REGION Network 61: UNIT 2 STATION 3 MEASURING RESET METHOD WORKING OR BLOCKED ALARM
   RUNG wire#powerrail
      Contact( "DB16337_U2_STA3_MEAS_RESET_TRIG".Done )
      I_Contact( "DB16004_U2_STA3_MEAS_CLIENT_INTERFACE".U02_STA3_MEAS_Method."Trigger reset".Outputs.Result )
      wire#w1
      Contact( "DB7256_UNIT_2_STA_3_MEAS_ENABLE_DISABLE".ENABLED )
      wire#w2
      Coil( "DB16000_OPC_UA_TRIGGER_ALARM".CLIENT.U2_STA3_MEAS.ALARMS.RESET_METHOD_WORKING_BLOCKED_A )
   END_RUNG
   RUNG wire#powerrail
      Contact( "DB16000_OPC_UA_TRIGGER_ALARM".CLIENT.U2_STA3_MEAS.ALARMS.RESET_METHOD_WORKING_BLOCKED_A )
      I_Contact( "DB2120_MPP_ITC_IPC".RESET_FAULTS )
   END_RUNG wire#w1
   RUNG wire#w2
      Coil( "DB426_ALARMS_WARNINGS".ALARMS.UNIT_02.STATION_3_MEASURING."720731" )
   END_RUNG
   // the same network as SCL:
   "DB16000_OPC_UA_TRIGGER_ALARM".CLIENT.U2_STA3_MEAS.ALARMS.RESET_METHOD_WORKING_BLOCKED_A := (("DB16337_U2_STA3_MEAS_RESET_TRIG".Done AND NOT "DB16004_U2_STA3_MEAS_CLIENT_INTERFACE".U02_STA3_MEAS_Method."Trigger reset".Outputs.Result) OR ("DB16000_OPC_UA_TRIGGER_ALARM".CLIENT.U2_STA3_MEAS.ALARMS.RESET_METHOD_WORKING_BLOCKED_A AND NOT "DB2120_MPP_ITC_IPC".RESET_FAULTS)) AND "DB7256_UNIT_2_STA_3_MEAS_ENABLE_DISABLE".ENABLED;
   "DB426_ALARMS_WARNINGS".ALARMS.UNIT_02.STATION_3_MEASURING."720731" := "DB16000_OPC_UA_TRIGGER_ALARM".CLIENT.U2_STA3_MEAS.ALARMS.RESET_METHOD_WORKING_BLOCKED_A;
END_REGION

REGION Network 62: UNIT 2 STATION 3 MEASURING READ VARIABLES CONNECTION ALARM
   RUNG wire#powerrail
      Contact( "DB16330_READLIST_U2_STA3_MEAS".Error )
      wire#w1
      Contact( "DB7256_UNIT_2_STA_3_MEAS_ENABLE_DISABLE".ENABLED )
      wire#w2
      Coil( "DB16000_OPC_UA_TRIGGER_ALARM".CLIENT.U2_STA3_MEAS.ALARMS.READ_VAR_CONNECTION_A )
   END_RUNG
   RUNG wire#powerrail
      Contact( "DB16000_OPC_UA_TRIGGER_ALARM".CLIENT.U2_STA3_MEAS.ALARMS.READ_VAR_CONNECTION_A )
      I_Contact( "DB2120_MPP_ITC_IPC".RESET_FAULTS )
   END_RUNG wire#w1
   RUNG wire#w2
      Coil( "DB426_ALARMS_WARNINGS".ALARMS.UNIT_02.STATION_3_MEASURING."720738" )
   END_RUNG
   // the same network as SCL:
   "DB16000_OPC_UA_TRIGGER_ALARM".CLIENT.U2_STA3_MEAS.ALARMS.READ_VAR_CONNECTION_A := ("DB16330_READLIST_U2_STA3_MEAS".Error OR ("DB16000_OPC_UA_TRIGGER_ALARM".CLIENT.U2_STA3_MEAS.ALARMS.READ_VAR_CONNECTION_A AND NOT "DB2120_MPP_ITC_IPC".RESET_FAULTS)) AND "DB7256_UNIT_2_STA_3_MEAS_ENABLE_DISABLE".ENABLED;
   "DB426_ALARMS_WARNINGS".ALARMS.UNIT_02.STATION_3_MEASURING."720738" := "DB16000_OPC_UA_TRIGGER_ALARM".CLIENT.U2_STA3_MEAS.ALARMS.READ_VAR_CONNECTION_A;
END_REGION

REGION Network 63: UNIT 2 STATION 3 MEASURING READ VARIABLES WORKING OR BLOCKED ALARM
   RUNG wire#powerrail
      Contact( "DB16330_READLIST_U2_STA3_MEAS".Done )
      Contact( "M_DUMMY_OFF" )
      wire#w1
      Contact( "DB7256_UNIT_2_STA_3_MEAS_ENABLE_DISABLE".ENABLED )
      wire#w2
      Coil( "DB16000_OPC_UA_TRIGGER_ALARM".CLIENT.U2_STA3_MEAS.ALARMS.READ_VAR_METHOD_WORKING_BLOCKED_A )
   END_RUNG
   RUNG wire#powerrail
      Contact( "DB16000_OPC_UA_TRIGGER_ALARM".CLIENT.U2_STA3_MEAS.ALARMS.READ_VAR_METHOD_WORKING_BLOCKED_A )
      I_Contact( "DB2120_MPP_ITC_IPC".RESET_FAULTS )
   END_RUNG wire#w1
   RUNG wire#w2
      Coil( "DB426_ALARMS_WARNINGS".ALARMS.UNIT_02.STATION_3_MEASURING."720739" )
   END_RUNG
   // the same network as SCL:
   "DB16000_OPC_UA_TRIGGER_ALARM".CLIENT.U2_STA3_MEAS.ALARMS.READ_VAR_METHOD_WORKING_BLOCKED_A := (("DB16330_READLIST_U2_STA3_MEAS".Done AND "M_DUMMY_OFF") OR ("DB16000_OPC_UA_TRIGGER_ALARM".CLIENT.U2_STA3_MEAS.ALARMS.READ_VAR_METHOD_WORKING_BLOCKED_A AND NOT "DB2120_MPP_ITC_IPC".RESET_FAULTS)) AND "DB7256_UNIT_2_STA_3_MEAS_ENABLE_DISABLE".ENABLED;
   "DB426_ALARMS_WARNINGS".ALARMS.UNIT_02.STATION_3_MEASURING."720739" := "DB16000_OPC_UA_TRIGGER_ALARM".CLIENT.U2_STA3_MEAS.ALARMS.READ_VAR_METHOD_WORKING_BLOCKED_A;
END_REGION

REGION Network 64: UNIT 2 STATION 3 MEASURING PROFILER CONFIGURATION ALARM
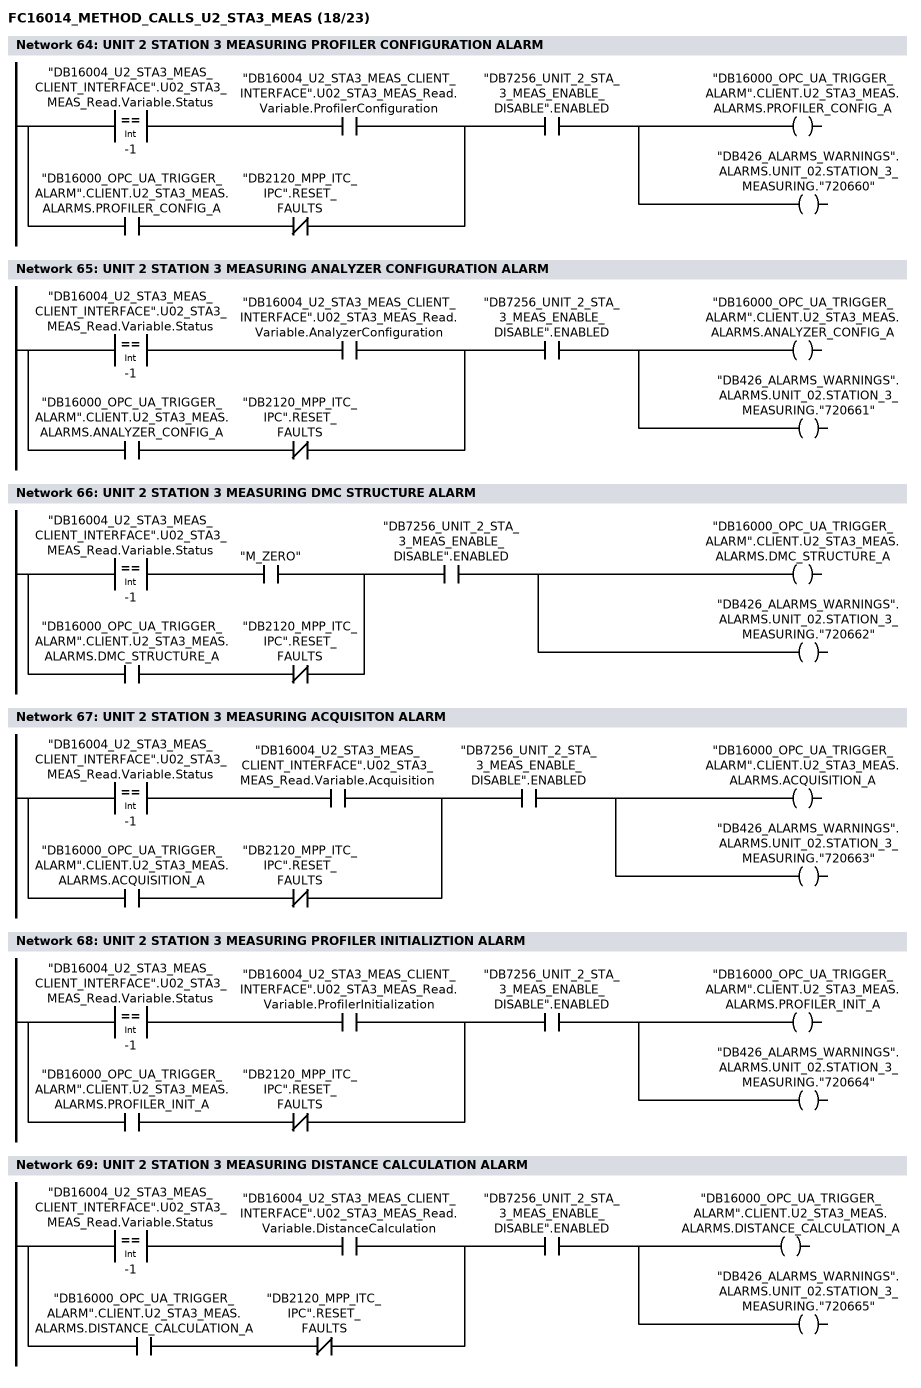
   RUNG wire#powerrail
      { S7_Templates := "SrcType := Int" } EQ_Contact(in1 := "DB16004_U2_STA3_MEAS_CLIENT_INTERFACE".U02_STA3_MEAS_Read.Variable.Status, in2 := -1)
      Contact( "DB16004_U2_STA3_MEAS_CLIENT_INTERFACE".U02_STA3_MEAS_Read.Variable.ProfilerConfiguration )
      wire#w1
      Contact( "DB7256_UNIT_2_STA_3_MEAS_ENABLE_DISABLE".ENABLED )
      wire#w2
      Coil( "DB16000_OPC_UA_TRIGGER_ALARM".CLIENT.U2_STA3_MEAS.ALARMS.PROFILER_CONFIG_A )
   END_RUNG
   RUNG wire#powerrail
      Contact( "DB16000_OPC_UA_TRIGGER_ALARM".CLIENT.U2_STA3_MEAS.ALARMS.PROFILER_CONFIG_A )
      I_Contact( "DB2120_MPP_ITC_IPC".RESET_FAULTS )
   END_RUNG wire#w1
   RUNG wire#w2
      Coil( "DB426_ALARMS_WARNINGS".ALARMS.UNIT_02.STATION_3_MEASURING."720660" )
   END_RUNG
   // the same network as SCL:
   "DB16000_OPC_UA_TRIGGER_ALARM".CLIENT.U2_STA3_MEAS.ALARMS.PROFILER_CONFIG_A := ((("DB16004_U2_STA3_MEAS_CLIENT_INTERFACE".U02_STA3_MEAS_Read.Variable.Status = (-1)) AND "DB16004_U2_STA3_MEAS_CLIENT_INTERFACE".U02_STA3_MEAS_Read.Variable.ProfilerConfiguration) OR ("DB16000_OPC_UA_TRIGGER_ALARM".CLIENT.U2_STA3_MEAS.ALARMS.PROFILER_CONFIG_A AND NOT "DB2120_MPP_ITC_IPC".RESET_FAULTS)) AND "DB7256_UNIT_2_STA_3_MEAS_ENABLE_DISABLE".ENABLED;
   "DB426_ALARMS_WARNINGS".ALARMS.UNIT_02.STATION_3_MEASURING."720660" := "DB16000_OPC_UA_TRIGGER_ALARM".CLIENT.U2_STA3_MEAS.ALARMS.PROFILER_CONFIG_A;
END_REGION

REGION Network 65: UNIT 2 STATION 3 MEASURING ANALYZER CONFIGURATION ALARM
   RUNG wire#powerrail
      { S7_Templates := "SrcType := Int" } EQ_Contact(in1 := "DB16004_U2_STA3_MEAS_CLIENT_INTERFACE".U02_STA3_MEAS_Read.Variable.Status, in2 := -1)
      Contact( "DB16004_U2_STA3_MEAS_CLIENT_INTERFACE".U02_STA3_MEAS_Read.Variable.AnalyzerConfiguration )
      wire#w1
      Contact( "DB7256_UNIT_2_STA_3_MEAS_ENABLE_DISABLE".ENABLED )
      wire#w2
      Coil( "DB16000_OPC_UA_TRIGGER_ALARM".CLIENT.U2_STA3_MEAS.ALARMS.ANALYZER_CONFIG_A )
   END_RUNG
   RUNG wire#powerrail
      Contact( "DB16000_OPC_UA_TRIGGER_ALARM".CLIENT.U2_STA3_MEAS.ALARMS.ANALYZER_CONFIG_A )
      I_Contact( "DB2120_MPP_ITC_IPC".RESET_FAULTS )
   END_RUNG wire#w1
   RUNG wire#w2
      Coil( "DB426_ALARMS_WARNINGS".ALARMS.UNIT_02.STATION_3_MEASURING."720661" )
   END_RUNG
   // the same network as SCL:
   "DB16000_OPC_UA_TRIGGER_ALARM".CLIENT.U2_STA3_MEAS.ALARMS.ANALYZER_CONFIG_A := ((("DB16004_U2_STA3_MEAS_CLIENT_INTERFACE".U02_STA3_MEAS_Read.Variable.Status = (-1)) AND "DB16004_U2_STA3_MEAS_CLIENT_INTERFACE".U02_STA3_MEAS_Read.Variable.AnalyzerConfiguration) OR ("DB16000_OPC_UA_TRIGGER_ALARM".CLIENT.U2_STA3_MEAS.ALARMS.ANALYZER_CONFIG_A AND NOT "DB2120_MPP_ITC_IPC".RESET_FAULTS)) AND "DB7256_UNIT_2_STA_3_MEAS_ENABLE_DISABLE".ENABLED;
   "DB426_ALARMS_WARNINGS".ALARMS.UNIT_02.STATION_3_MEASURING."720661" := "DB16000_OPC_UA_TRIGGER_ALARM".CLIENT.U2_STA3_MEAS.ALARMS.ANALYZER_CONFIG_A;
END_REGION

REGION Network 66: UNIT 2 STATION 3 MEASURING DMC STRUCTURE ALARM
   RUNG wire#powerrail
      { S7_Templates := "SrcType := Int" } EQ_Contact(in1 := "DB16004_U2_STA3_MEAS_CLIENT_INTERFACE".U02_STA3_MEAS_Read.Variable.Status, in2 := -1)
      Contact( "M_ZERO" )
      wire#w1
      Contact( "DB7256_UNIT_2_STA_3_MEAS_ENABLE_DISABLE".ENABLED )
      wire#w2
      Coil( "DB16000_OPC_UA_TRIGGER_ALARM".CLIENT.U2_STA3_MEAS.ALARMS.DMC_STRUCTURE_A )
   END_RUNG
   RUNG wire#powerrail
      Contact( "DB16000_OPC_UA_TRIGGER_ALARM".CLIENT.U2_STA3_MEAS.ALARMS.DMC_STRUCTURE_A )
      I_Contact( "DB2120_MPP_ITC_IPC".RESET_FAULTS )
   END_RUNG wire#w1
   RUNG wire#w2
      Coil( "DB426_ALARMS_WARNINGS".ALARMS.UNIT_02.STATION_3_MEASURING."720662" )
   END_RUNG
   // the same network as SCL:
   "DB16000_OPC_UA_TRIGGER_ALARM".CLIENT.U2_STA3_MEAS.ALARMS.DMC_STRUCTURE_A := ((("DB16004_U2_STA3_MEAS_CLIENT_INTERFACE".U02_STA3_MEAS_Read.Variable.Status = (-1)) AND "M_ZERO") OR ("DB16000_OPC_UA_TRIGGER_ALARM".CLIENT.U2_STA3_MEAS.ALARMS.DMC_STRUCTURE_A AND NOT "DB2120_MPP_ITC_IPC".RESET_FAULTS)) AND "DB7256_UNIT_2_STA_3_MEAS_ENABLE_DISABLE".ENABLED;
   "DB426_ALARMS_WARNINGS".ALARMS.UNIT_02.STATION_3_MEASURING."720662" := "DB16000_OPC_UA_TRIGGER_ALARM".CLIENT.U2_STA3_MEAS.ALARMS.DMC_STRUCTURE_A;
END_REGION

REGION Network 67: UNIT 2 STATION 3 MEASURING ACQUISITON ALARM
   RUNG wire#powerrail
      { S7_Templates := "SrcType := Int" } EQ_Contact(in1 := "DB16004_U2_STA3_MEAS_CLIENT_INTERFACE".U02_STA3_MEAS_Read.Variable.Status, in2 := -1)
      Contact( "DB16004_U2_STA3_MEAS_CLIENT_INTERFACE".U02_STA3_MEAS_Read.Variable.Acquisition )
      wire#w1
      Contact( "DB7256_UNIT_2_STA_3_MEAS_ENABLE_DISABLE".ENABLED )
      wire#w2
      Coil( "DB16000_OPC_UA_TRIGGER_ALARM".CLIENT.U2_STA3_MEAS.ALARMS.ACQUISITION_A )
   END_RUNG
   RUNG wire#powerrail
      Contact( "DB16000_OPC_UA_TRIGGER_ALARM".CLIENT.U2_STA3_MEAS.ALARMS.ACQUISITION_A )
      I_Contact( "DB2120_MPP_ITC_IPC".RESET_FAULTS )
   END_RUNG wire#w1
   RUNG wire#w2
      Coil( "DB426_ALARMS_WARNINGS".ALARMS.UNIT_02.STATION_3_MEASURING."720663" )
   END_RUNG
   // the same network as SCL:
   "DB16000_OPC_UA_TRIGGER_ALARM".CLIENT.U2_STA3_MEAS.ALARMS.ACQUISITION_A := ((("DB16004_U2_STA3_MEAS_CLIENT_INTERFACE".U02_STA3_MEAS_Read.Variable.Status = (-1)) AND "DB16004_U2_STA3_MEAS_CLIENT_INTERFACE".U02_STA3_MEAS_Read.Variable.Acquisition) OR ("DB16000_OPC_UA_TRIGGER_ALARM".CLIENT.U2_STA3_MEAS.ALARMS.ACQUISITION_A AND NOT "DB2120_MPP_ITC_IPC".RESET_FAULTS)) AND "DB7256_UNIT_2_STA_3_MEAS_ENABLE_DISABLE".ENABLED;
   "DB426_ALARMS_WARNINGS".ALARMS.UNIT_02.STATION_3_MEASURING."720663" := "DB16000_OPC_UA_TRIGGER_ALARM".CLIENT.U2_STA3_MEAS.ALARMS.ACQUISITION_A;
END_REGION

REGION Network 68: UNIT 2 STATION 3 MEASURING PROFILER INITIALIZTION ALARM
   RUNG wire#powerrail
      { S7_Templates := "SrcType := Int" } EQ_Contact(in1 := "DB16004_U2_STA3_MEAS_CLIENT_INTERFACE".U02_STA3_MEAS_Read.Variable.Status, in2 := -1)
      Contact( "DB16004_U2_STA3_MEAS_CLIENT_INTERFACE".U02_STA3_MEAS_Read.Variable.ProfilerInitialization )
      wire#w1
      Contact( "DB7256_UNIT_2_STA_3_MEAS_ENABLE_DISABLE".ENABLED )
      wire#w2
      Coil( "DB16000_OPC_UA_TRIGGER_ALARM".CLIENT.U2_STA3_MEAS.ALARMS.PROFILER_INIT_A )
   END_RUNG
   RUNG wire#powerrail
      Contact( "DB16000_OPC_UA_TRIGGER_ALARM".CLIENT.U2_STA3_MEAS.ALARMS.PROFILER_INIT_A )
      I_Contact( "DB2120_MPP_ITC_IPC".RESET_FAULTS )
   END_RUNG wire#w1
   RUNG wire#w2
      Coil( "DB426_ALARMS_WARNINGS".ALARMS.UNIT_02.STATION_3_MEASURING."720664" )
   END_RUNG
   // the same network as SCL:
   "DB16000_OPC_UA_TRIGGER_ALARM".CLIENT.U2_STA3_MEAS.ALARMS.PROFILER_INIT_A := ((("DB16004_U2_STA3_MEAS_CLIENT_INTERFACE".U02_STA3_MEAS_Read.Variable.Status = (-1)) AND "DB16004_U2_STA3_MEAS_CLIENT_INTERFACE".U02_STA3_MEAS_Read.Variable.ProfilerInitialization) OR ("DB16000_OPC_UA_TRIGGER_ALARM".CLIENT.U2_STA3_MEAS.ALARMS.PROFILER_INIT_A AND NOT "DB2120_MPP_ITC_IPC".RESET_FAULTS)) AND "DB7256_UNIT_2_STA_3_MEAS_ENABLE_DISABLE".ENABLED;
   "DB426_ALARMS_WARNINGS".ALARMS.UNIT_02.STATION_3_MEASURING."720664" := "DB16000_OPC_UA_TRIGGER_ALARM".CLIENT.U2_STA3_MEAS.ALARMS.PROFILER_INIT_A;
END_REGION

REGION Network 69: UNIT 2 STATION 3 MEASURING DISTANCE CALCULATION ALARM
   RUNG wire#powerrail
      { S7_Templates := "SrcType := Int" } EQ_Contact(in1 := "DB16004_U2_STA3_MEAS_CLIENT_INTERFACE".U02_STA3_MEAS_Read.Variable.Status, in2 := -1)
      Contact( "DB16004_U2_STA3_MEAS_CLIENT_INTERFACE".U02_STA3_MEAS_Read.Variable.DistanceCalculation )
      wire#w1
      Contact( "DB7256_UNIT_2_STA_3_MEAS_ENABLE_DISABLE".ENABLED )
      wire#w2
      Coil( "DB16000_OPC_UA_TRIGGER_ALARM".CLIENT.U2_STA3_MEAS.ALARMS.DISTANCE_CALCULATION_A )
   END_RUNG
   RUNG wire#powerrail
      Contact( "DB16000_OPC_UA_TRIGGER_ALARM".CLIENT.U2_STA3_MEAS.ALARMS.DISTANCE_CALCULATION_A )
      I_Contact( "DB2120_MPP_ITC_IPC".RESET_FAULTS )
   END_RUNG wire#w1
   RUNG wire#w2
      Coil( "DB426_ALARMS_WARNINGS".ALARMS.UNIT_02.STATION_3_MEASURING."720665" )
   END_RUNG
   // the same network as SCL:
   "DB16000_OPC_UA_TRIGGER_ALARM".CLIENT.U2_STA3_MEAS.ALARMS.DISTANCE_CALCULATION_A := ((("DB16004_U2_STA3_MEAS_CLIENT_INTERFACE".U02_STA3_MEAS_Read.Variable.Status = (-1)) AND "DB16004_U2_STA3_MEAS_CLIENT_INTERFACE".U02_STA3_MEAS_Read.Variable.DistanceCalculation) OR ("DB16000_OPC_UA_TRIGGER_ALARM".CLIENT.U2_STA3_MEAS.ALARMS.DISTANCE_CALCULATION_A AND NOT "DB2120_MPP_ITC_IPC".RESET_FAULTS)) AND "DB7256_UNIT_2_STA_3_MEAS_ENABLE_DISABLE".ENABLED;
   "DB426_ALARMS_WARNINGS".ALARMS.UNIT_02.STATION_3_MEASURING."720665" := "DB16000_OPC_UA_TRIGGER_ALARM".CLIENT.U2_STA3_MEAS.ALARMS.DISTANCE_CALCULATION_A;
END_REGION

REGION Network 70: UNIT 2 STATION 3 MEASURING LAYER GROWTH ANALYSIS ALARM
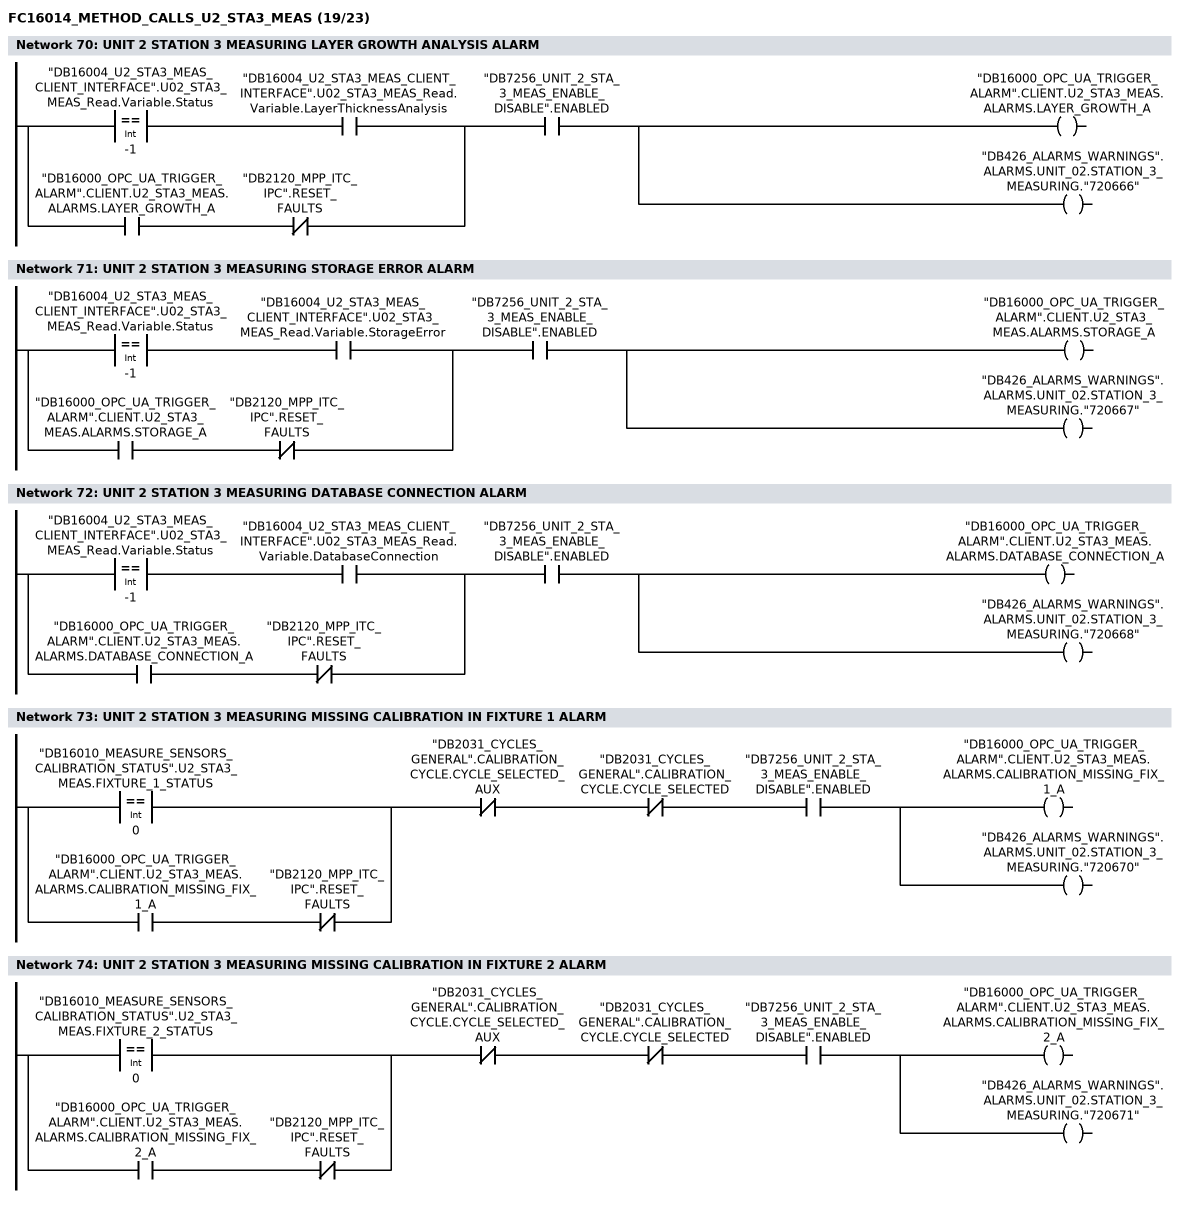
   RUNG wire#powerrail
      { S7_Templates := "SrcType := Int" } EQ_Contact(in1 := "DB16004_U2_STA3_MEAS_CLIENT_INTERFACE".U02_STA3_MEAS_Read.Variable.Status, in2 := -1)
      Contact( "DB16004_U2_STA3_MEAS_CLIENT_INTERFACE".U02_STA3_MEAS_Read.Variable.LayerThicknessAnalysis )
      wire#w1
      Contact( "DB7256_UNIT_2_STA_3_MEAS_ENABLE_DISABLE".ENABLED )
      wire#w2
      Coil( "DB16000_OPC_UA_TRIGGER_ALARM".CLIENT.U2_STA3_MEAS.ALARMS.LAYER_GROWTH_A )
   END_RUNG
   RUNG wire#powerrail
      Contact( "DB16000_OPC_UA_TRIGGER_ALARM".CLIENT.U2_STA3_MEAS.ALARMS.LAYER_GROWTH_A )
      I_Contact( "DB2120_MPP_ITC_IPC".RESET_FAULTS )
   END_RUNG wire#w1
   RUNG wire#w2
      Coil( "DB426_ALARMS_WARNINGS".ALARMS.UNIT_02.STATION_3_MEASURING."720666" )
   END_RUNG
   // the same network as SCL:
   "DB16000_OPC_UA_TRIGGER_ALARM".CLIENT.U2_STA3_MEAS.ALARMS.LAYER_GROWTH_A := ((("DB16004_U2_STA3_MEAS_CLIENT_INTERFACE".U02_STA3_MEAS_Read.Variable.Status = (-1)) AND "DB16004_U2_STA3_MEAS_CLIENT_INTERFACE".U02_STA3_MEAS_Read.Variable.LayerThicknessAnalysis) OR ("DB16000_OPC_UA_TRIGGER_ALARM".CLIENT.U2_STA3_MEAS.ALARMS.LAYER_GROWTH_A AND NOT "DB2120_MPP_ITC_IPC".RESET_FAULTS)) AND "DB7256_UNIT_2_STA_3_MEAS_ENABLE_DISABLE".ENABLED;
   "DB426_ALARMS_WARNINGS".ALARMS.UNIT_02.STATION_3_MEASURING."720666" := "DB16000_OPC_UA_TRIGGER_ALARM".CLIENT.U2_STA3_MEAS.ALARMS.LAYER_GROWTH_A;
END_REGION

REGION Network 71: UNIT 2 STATION 3 MEASURING STORAGE ERROR ALARM
   RUNG wire#powerrail
      { S7_Templates := "SrcType := Int" } EQ_Contact(in1 := "DB16004_U2_STA3_MEAS_CLIENT_INTERFACE".U02_STA3_MEAS_Read.Variable.Status, in2 := -1)
      Contact( "DB16004_U2_STA3_MEAS_CLIENT_INTERFACE".U02_STA3_MEAS_Read.Variable.StorageError )
      wire#w1
      Contact( "DB7256_UNIT_2_STA_3_MEAS_ENABLE_DISABLE".ENABLED )
      wire#w2
      Coil( "DB16000_OPC_UA_TRIGGER_ALARM".CLIENT.U2_STA3_MEAS.ALARMS.STORAGE_A )
   END_RUNG
   RUNG wire#powerrail
      Contact( "DB16000_OPC_UA_TRIGGER_ALARM".CLIENT.U2_STA3_MEAS.ALARMS.STORAGE_A )
      I_Contact( "DB2120_MPP_ITC_IPC".RESET_FAULTS )
   END_RUNG wire#w1
   RUNG wire#w2
      Coil( "DB426_ALARMS_WARNINGS".ALARMS.UNIT_02.STATION_3_MEASURING."720667" )
   END_RUNG
   // the same network as SCL:
   "DB16000_OPC_UA_TRIGGER_ALARM".CLIENT.U2_STA3_MEAS.ALARMS.STORAGE_A := ((("DB16004_U2_STA3_MEAS_CLIENT_INTERFACE".U02_STA3_MEAS_Read.Variable.Status = (-1)) AND "DB16004_U2_STA3_MEAS_CLIENT_INTERFACE".U02_STA3_MEAS_Read.Variable.StorageError) OR ("DB16000_OPC_UA_TRIGGER_ALARM".CLIENT.U2_STA3_MEAS.ALARMS.STORAGE_A AND NOT "DB2120_MPP_ITC_IPC".RESET_FAULTS)) AND "DB7256_UNIT_2_STA_3_MEAS_ENABLE_DISABLE".ENABLED;
   "DB426_ALARMS_WARNINGS".ALARMS.UNIT_02.STATION_3_MEASURING."720667" := "DB16000_OPC_UA_TRIGGER_ALARM".CLIENT.U2_STA3_MEAS.ALARMS.STORAGE_A;
END_REGION

REGION Network 72: UNIT 2 STATION 3 MEASURING DATABASE CONNECTION ALARM
   RUNG wire#powerrail
      { S7_Templates := "SrcType := Int" } EQ_Contact(in1 := "DB16004_U2_STA3_MEAS_CLIENT_INTERFACE".U02_STA3_MEAS_Read.Variable.Status, in2 := -1)
      Contact( "DB16004_U2_STA3_MEAS_CLIENT_INTERFACE".U02_STA3_MEAS_Read.Variable.DatabaseConnection )
      wire#w1
      Contact( "DB7256_UNIT_2_STA_3_MEAS_ENABLE_DISABLE".ENABLED )
      wire#w2
      Coil( "DB16000_OPC_UA_TRIGGER_ALARM".CLIENT.U2_STA3_MEAS.ALARMS.DATABASE_CONNECTION_A )
   END_RUNG
   RUNG wire#powerrail
      Contact( "DB16000_OPC_UA_TRIGGER_ALARM".CLIENT.U2_STA3_MEAS.ALARMS.DATABASE_CONNECTION_A )
      I_Contact( "DB2120_MPP_ITC_IPC".RESET_FAULTS )
   END_RUNG wire#w1
   RUNG wire#w2
      Coil( "DB426_ALARMS_WARNINGS".ALARMS.UNIT_02.STATION_3_MEASURING."720668" )
   END_RUNG
   // the same network as SCL:
   "DB16000_OPC_UA_TRIGGER_ALARM".CLIENT.U2_STA3_MEAS.ALARMS.DATABASE_CONNECTION_A := ((("DB16004_U2_STA3_MEAS_CLIENT_INTERFACE".U02_STA3_MEAS_Read.Variable.Status = (-1)) AND "DB16004_U2_STA3_MEAS_CLIENT_INTERFACE".U02_STA3_MEAS_Read.Variable.DatabaseConnection) OR ("DB16000_OPC_UA_TRIGGER_ALARM".CLIENT.U2_STA3_MEAS.ALARMS.DATABASE_CONNECTION_A AND NOT "DB2120_MPP_ITC_IPC".RESET_FAULTS)) AND "DB7256_UNIT_2_STA_3_MEAS_ENABLE_DISABLE".ENABLED;
   "DB426_ALARMS_WARNINGS".ALARMS.UNIT_02.STATION_3_MEASURING."720668" := "DB16000_OPC_UA_TRIGGER_ALARM".CLIENT.U2_STA3_MEAS.ALARMS.DATABASE_CONNECTION_A;
END_REGION

REGION Network 73: UNIT 2 STATION 3 MEASURING MISSING CALIBRATION IN FIXTURE 1 ALARM
   RUNG wire#powerrail
      { S7_Templates := "SrcType := Int" } EQ_Contact(in1 := "DB16010_MEASURE_SENSORS_CALIBRATION_STATUS".U2_STA3_MEAS.FIXTURE_1_STATUS, in2 := 0)
      wire#w1
      I_Contact( "DB2031_CYCLES_GENERAL".CALIBRATION_CYCLE.CYCLE_SELECTED_AUX )
      I_Contact( "DB2031_CYCLES_GENERAL".CALIBRATION_CYCLE.CYCLE_SELECTED )
      Contact( "DB7256_UNIT_2_STA_3_MEAS_ENABLE_DISABLE".ENABLED )
      wire#w2
      Coil( "DB16000_OPC_UA_TRIGGER_ALARM".CLIENT.U2_STA3_MEAS.ALARMS.CALIBRATION_MISSING_FIX_1_A )
   END_RUNG
   RUNG wire#powerrail
      Contact( "DB16000_OPC_UA_TRIGGER_ALARM".CLIENT.U2_STA3_MEAS.ALARMS.CALIBRATION_MISSING_FIX_1_A )
      I_Contact( "DB2120_MPP_ITC_IPC".RESET_FAULTS )
   END_RUNG wire#w1
   RUNG wire#w2
      Coil( "DB426_ALARMS_WARNINGS".ALARMS.UNIT_02.STATION_3_MEASURING."720670" )
   END_RUNG
   // the same network as SCL:
   "DB16000_OPC_UA_TRIGGER_ALARM".CLIENT.U2_STA3_MEAS.ALARMS.CALIBRATION_MISSING_FIX_1_A := (("DB16010_MEASURE_SENSORS_CALIBRATION_STATUS".U2_STA3_MEAS.FIXTURE_1_STATUS = 0) OR ("DB16000_OPC_UA_TRIGGER_ALARM".CLIENT.U2_STA3_MEAS.ALARMS.CALIBRATION_MISSING_FIX_1_A AND NOT "DB2120_MPP_ITC_IPC".RESET_FAULTS)) AND NOT "DB2031_CYCLES_GENERAL".CALIBRATION_CYCLE.CYCLE_SELECTED_AUX AND NOT "DB2031_CYCLES_GENERAL".CALIBRATION_CYCLE.CYCLE_SELECTED AND "DB7256_UNIT_2_STA_3_MEAS_ENABLE_DISABLE".ENABLED;
   "DB426_ALARMS_WARNINGS".ALARMS.UNIT_02.STATION_3_MEASURING."720670" := "DB16000_OPC_UA_TRIGGER_ALARM".CLIENT.U2_STA3_MEAS.ALARMS.CALIBRATION_MISSING_FIX_1_A;
END_REGION

REGION Network 74: UNIT 2 STATION 3 MEASURING MISSING CALIBRATION IN FIXTURE 2 ALARM
   RUNG wire#powerrail
      { S7_Templates := "SrcType := Int" } EQ_Contact(in1 := "DB16010_MEASURE_SENSORS_CALIBRATION_STATUS".U2_STA3_MEAS.FIXTURE_2_STATUS, in2 := 0)
      wire#w1
      I_Contact( "DB2031_CYCLES_GENERAL".CALIBRATION_CYCLE.CYCLE_SELECTED_AUX )
      I_Contact( "DB2031_CYCLES_GENERAL".CALIBRATION_CYCLE.CYCLE_SELECTED )
      Contact( "DB7256_UNIT_2_STA_3_MEAS_ENABLE_DISABLE".ENABLED )
      wire#w2
      Coil( "DB16000_OPC_UA_TRIGGER_ALARM".CLIENT.U2_STA3_MEAS.ALARMS.CALIBRATION_MISSING_FIX_2_A )
   END_RUNG
   RUNG wire#powerrail
      Contact( "DB16000_OPC_UA_TRIGGER_ALARM".CLIENT.U2_STA3_MEAS.ALARMS.CALIBRATION_MISSING_FIX_2_A )
      I_Contact( "DB2120_MPP_ITC_IPC".RESET_FAULTS )
   END_RUNG wire#w1
   RUNG wire#w2
      Coil( "DB426_ALARMS_WARNINGS".ALARMS.UNIT_02.STATION_3_MEASURING."720671" )
   END_RUNG
   // the same network as SCL:
   "DB16000_OPC_UA_TRIGGER_ALARM".CLIENT.U2_STA3_MEAS.ALARMS.CALIBRATION_MISSING_FIX_2_A := (("DB16010_MEASURE_SENSORS_CALIBRATION_STATUS".U2_STA3_MEAS.FIXTURE_2_STATUS = 0) OR ("DB16000_OPC_UA_TRIGGER_ALARM".CLIENT.U2_STA3_MEAS.ALARMS.CALIBRATION_MISSING_FIX_2_A AND NOT "DB2120_MPP_ITC_IPC".RESET_FAULTS)) AND NOT "DB2031_CYCLES_GENERAL".CALIBRATION_CYCLE.CYCLE_SELECTED_AUX AND NOT "DB2031_CYCLES_GENERAL".CALIBRATION_CYCLE.CYCLE_SELECTED AND "DB7256_UNIT_2_STA_3_MEAS_ENABLE_DISABLE".ENABLED;
   "DB426_ALARMS_WARNINGS".ALARMS.UNIT_02.STATION_3_MEASURING."720671" := "DB16000_OPC_UA_TRIGGER_ALARM".CLIENT.U2_STA3_MEAS.ALARMS.CALIBRATION_MISSING_FIX_2_A;
END_REGION

REGION Network 75: UNIT 2 STATION 3 MEASURING MISSING CALIBRATION IN FIXTURE 3 ALARM
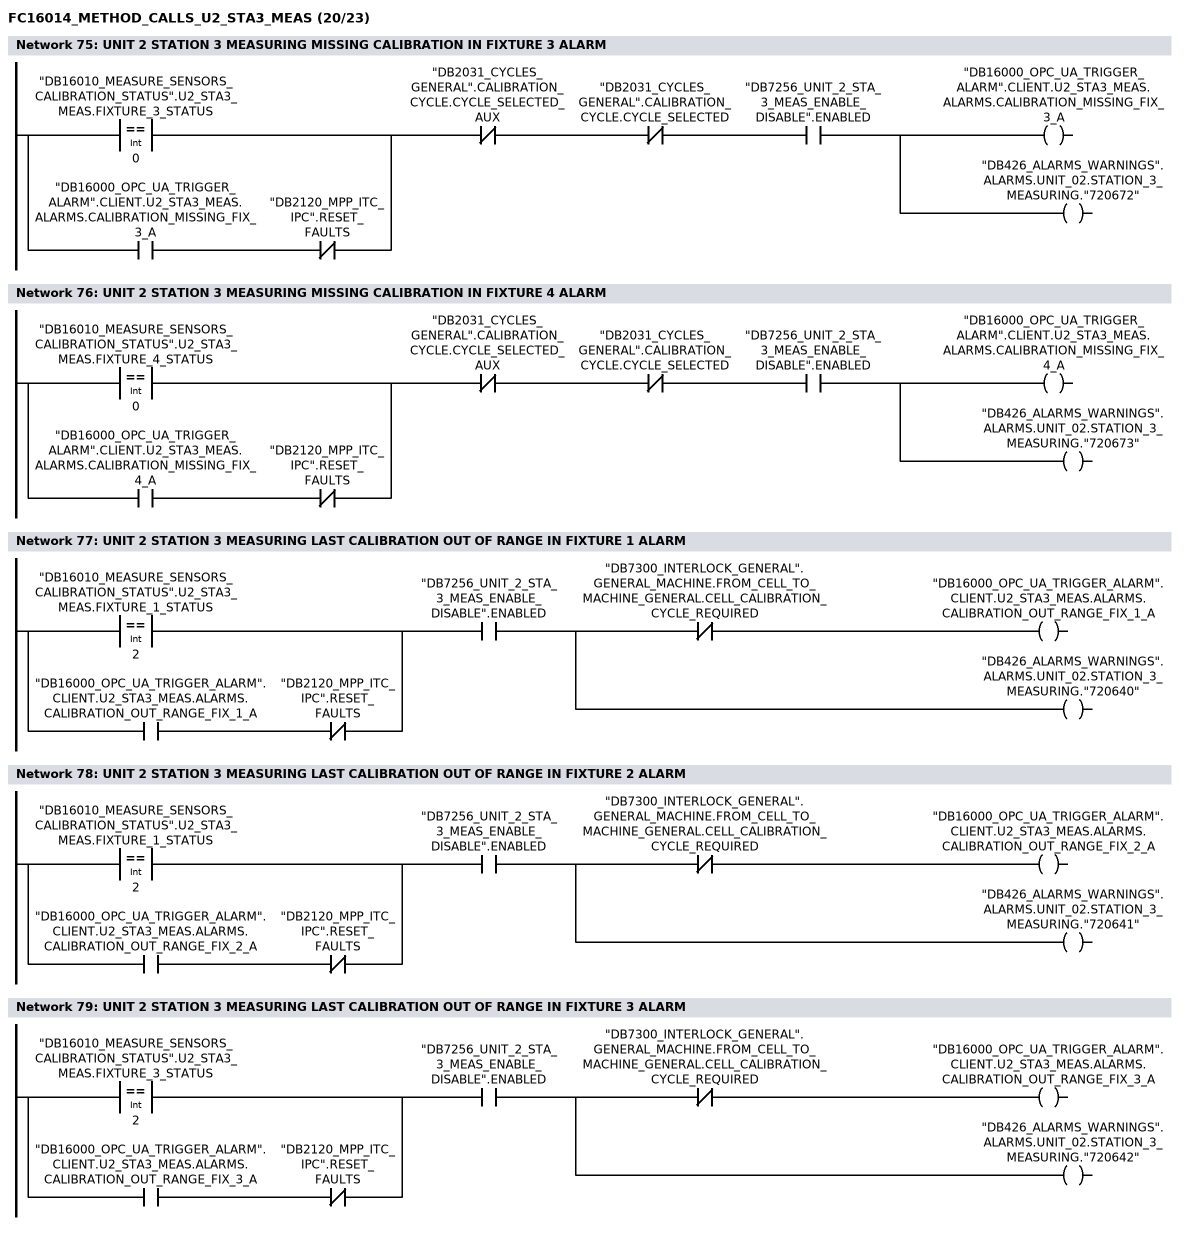
   RUNG wire#powerrail
      { S7_Templates := "SrcType := Int" } EQ_Contact(in1 := "DB16010_MEASURE_SENSORS_CALIBRATION_STATUS".U2_STA3_MEAS.FIXTURE_3_STATUS, in2 := 0)
      wire#w1
      I_Contact( "DB2031_CYCLES_GENERAL".CALIBRATION_CYCLE.CYCLE_SELECTED_AUX )
      I_Contact( "DB2031_CYCLES_GENERAL".CALIBRATION_CYCLE.CYCLE_SELECTED )
      Contact( "DB7256_UNIT_2_STA_3_MEAS_ENABLE_DISABLE".ENABLED )
      wire#w2
      Coil( "DB16000_OPC_UA_TRIGGER_ALARM".CLIENT.U2_STA3_MEAS.ALARMS.CALIBRATION_MISSING_FIX_3_A )
   END_RUNG
   RUNG wire#powerrail
      Contact( "DB16000_OPC_UA_TRIGGER_ALARM".CLIENT.U2_STA3_MEAS.ALARMS.CALIBRATION_MISSING_FIX_3_A )
      I_Contact( "DB2120_MPP_ITC_IPC".RESET_FAULTS )
   END_RUNG wire#w1
   RUNG wire#w2
      Coil( "DB426_ALARMS_WARNINGS".ALARMS.UNIT_02.STATION_3_MEASURING."720672" )
   END_RUNG
   // the same network as SCL:
   "DB16000_OPC_UA_TRIGGER_ALARM".CLIENT.U2_STA3_MEAS.ALARMS.CALIBRATION_MISSING_FIX_3_A := (("DB16010_MEASURE_SENSORS_CALIBRATION_STATUS".U2_STA3_MEAS.FIXTURE_3_STATUS = 0) OR ("DB16000_OPC_UA_TRIGGER_ALARM".CLIENT.U2_STA3_MEAS.ALARMS.CALIBRATION_MISSING_FIX_3_A AND NOT "DB2120_MPP_ITC_IPC".RESET_FAULTS)) AND NOT "DB2031_CYCLES_GENERAL".CALIBRATION_CYCLE.CYCLE_SELECTED_AUX AND NOT "DB2031_CYCLES_GENERAL".CALIBRATION_CYCLE.CYCLE_SELECTED AND "DB7256_UNIT_2_STA_3_MEAS_ENABLE_DISABLE".ENABLED;
   "DB426_ALARMS_WARNINGS".ALARMS.UNIT_02.STATION_3_MEASURING."720672" := "DB16000_OPC_UA_TRIGGER_ALARM".CLIENT.U2_STA3_MEAS.ALARMS.CALIBRATION_MISSING_FIX_3_A;
END_REGION

REGION Network 76: UNIT 2 STATION 3 MEASURING MISSING CALIBRATION IN FIXTURE 4 ALARM
   RUNG wire#powerrail
      { S7_Templates := "SrcType := Int" } EQ_Contact(in1 := "DB16010_MEASURE_SENSORS_CALIBRATION_STATUS".U2_STA3_MEAS.FIXTURE_4_STATUS, in2 := 0)
      wire#w1
      I_Contact( "DB2031_CYCLES_GENERAL".CALIBRATION_CYCLE.CYCLE_SELECTED_AUX )
      I_Contact( "DB2031_CYCLES_GENERAL".CALIBRATION_CYCLE.CYCLE_SELECTED )
      Contact( "DB7256_UNIT_2_STA_3_MEAS_ENABLE_DISABLE".ENABLED )
      wire#w2
      Coil( "DB16000_OPC_UA_TRIGGER_ALARM".CLIENT.U2_STA3_MEAS.ALARMS.CALIBRATION_MISSING_FIX_4_A )
   END_RUNG
   RUNG wire#powerrail
      Contact( "DB16000_OPC_UA_TRIGGER_ALARM".CLIENT.U2_STA3_MEAS.ALARMS.CALIBRATION_MISSING_FIX_4_A )
      I_Contact( "DB2120_MPP_ITC_IPC".RESET_FAULTS )
   END_RUNG wire#w1
   RUNG wire#w2
      Coil( "DB426_ALARMS_WARNINGS".ALARMS.UNIT_02.STATION_3_MEASURING."720673" )
   END_RUNG
   // the same network as SCL:
   "DB16000_OPC_UA_TRIGGER_ALARM".CLIENT.U2_STA3_MEAS.ALARMS.CALIBRATION_MISSING_FIX_4_A := (("DB16010_MEASURE_SENSORS_CALIBRATION_STATUS".U2_STA3_MEAS.FIXTURE_4_STATUS = 0) OR ("DB16000_OPC_UA_TRIGGER_ALARM".CLIENT.U2_STA3_MEAS.ALARMS.CALIBRATION_MISSING_FIX_4_A AND NOT "DB2120_MPP_ITC_IPC".RESET_FAULTS)) AND NOT "DB2031_CYCLES_GENERAL".CALIBRATION_CYCLE.CYCLE_SELECTED_AUX AND NOT "DB2031_CYCLES_GENERAL".CALIBRATION_CYCLE.CYCLE_SELECTED AND "DB7256_UNIT_2_STA_3_MEAS_ENABLE_DISABLE".ENABLED;
   "DB426_ALARMS_WARNINGS".ALARMS.UNIT_02.STATION_3_MEASURING."720673" := "DB16000_OPC_UA_TRIGGER_ALARM".CLIENT.U2_STA3_MEAS.ALARMS.CALIBRATION_MISSING_FIX_4_A;
END_REGION

REGION Network 77: UNIT 2 STATION 3 MEASURING LAST CALIBRATION OUT OF RANGE IN FIXTURE 1 ALARM
   RUNG wire#powerrail
      { S7_Templates := "SrcType := Int" } EQ_Contact(in1 := "DB16010_MEASURE_SENSORS_CALIBRATION_STATUS".U2_STA3_MEAS.FIXTURE_1_STATUS, in2 := 2)
      wire#w1
      Contact( "DB7256_UNIT_2_STA_3_MEAS_ENABLE_DISABLE".ENABLED )
      wire#w2
      I_Contact( "DB7300_INTERLOCK_GENERAL".GENERAL_MACHINE.FROM_CELL_TO_MACHINE_GENERAL.CELL_CALIBRATION_CYCLE_REQUIRED )
      Coil( "DB16000_OPC_UA_TRIGGER_ALARM".CLIENT.U2_STA3_MEAS.ALARMS.CALIBRATION_OUT_RANGE_FIX_1_A )
   END_RUNG
   RUNG wire#powerrail
      Contact( "DB16000_OPC_UA_TRIGGER_ALARM".CLIENT.U2_STA3_MEAS.ALARMS.CALIBRATION_OUT_RANGE_FIX_1_A )
      I_Contact( "DB2120_MPP_ITC_IPC".RESET_FAULTS )
   END_RUNG wire#w1
   RUNG wire#w2
      Coil( "DB426_ALARMS_WARNINGS".ALARMS.UNIT_02.STATION_3_MEASURING."720640" )
   END_RUNG
   // the same network as SCL:
   #_w1 := (("DB16010_MEASURE_SENSORS_CALIBRATION_STATUS".U2_STA3_MEAS.FIXTURE_1_STATUS = 2) OR ("DB16000_OPC_UA_TRIGGER_ALARM".CLIENT.U2_STA3_MEAS.ALARMS.CALIBRATION_OUT_RANGE_FIX_1_A AND NOT "DB2120_MPP_ITC_IPC".RESET_FAULTS)) AND "DB7256_UNIT_2_STA_3_MEAS_ENABLE_DISABLE".ENABLED;
   "DB16000_OPC_UA_TRIGGER_ALARM".CLIENT.U2_STA3_MEAS.ALARMS.CALIBRATION_OUT_RANGE_FIX_1_A := #_w1 AND NOT "DB7300_INTERLOCK_GENERAL".GENERAL_MACHINE.FROM_CELL_TO_MACHINE_GENERAL.CELL_CALIBRATION_CYCLE_REQUIRED;
   "DB426_ALARMS_WARNINGS".ALARMS.UNIT_02.STATION_3_MEASURING."720640" := #_w1;
END_REGION

REGION Network 78: UNIT 2 STATION 3 MEASURING LAST CALIBRATION OUT OF RANGE IN FIXTURE 2 ALARM
   RUNG wire#powerrail
      { S7_Templates := "SrcType := Int" } EQ_Contact(in1 := "DB16010_MEASURE_SENSORS_CALIBRATION_STATUS".U2_STA3_MEAS.FIXTURE_1_STATUS, in2 := 2)
      wire#w1
      Contact( "DB7256_UNIT_2_STA_3_MEAS_ENABLE_DISABLE".ENABLED )
      wire#w2
      I_Contact( "DB7300_INTERLOCK_GENERAL".GENERAL_MACHINE.FROM_CELL_TO_MACHINE_GENERAL.CELL_CALIBRATION_CYCLE_REQUIRED )
      Coil( "DB16000_OPC_UA_TRIGGER_ALARM".CLIENT.U2_STA3_MEAS.ALARMS.CALIBRATION_OUT_RANGE_FIX_2_A )
   END_RUNG
   RUNG wire#powerrail
      Contact( "DB16000_OPC_UA_TRIGGER_ALARM".CLIENT.U2_STA3_MEAS.ALARMS.CALIBRATION_OUT_RANGE_FIX_2_A )
      I_Contact( "DB2120_MPP_ITC_IPC".RESET_FAULTS )
   END_RUNG wire#w1
   RUNG wire#w2
      Coil( "DB426_ALARMS_WARNINGS".ALARMS.UNIT_02.STATION_3_MEASURING."720641" )
   END_RUNG
   // the same network as SCL:
   #_w1 := (("DB16010_MEASURE_SENSORS_CALIBRATION_STATUS".U2_STA3_MEAS.FIXTURE_1_STATUS = 2) OR ("DB16000_OPC_UA_TRIGGER_ALARM".CLIENT.U2_STA3_MEAS.ALARMS.CALIBRATION_OUT_RANGE_FIX_2_A AND NOT "DB2120_MPP_ITC_IPC".RESET_FAULTS)) AND "DB7256_UNIT_2_STA_3_MEAS_ENABLE_DISABLE".ENABLED;
   "DB16000_OPC_UA_TRIGGER_ALARM".CLIENT.U2_STA3_MEAS.ALARMS.CALIBRATION_OUT_RANGE_FIX_2_A := #_w1 AND NOT "DB7300_INTERLOCK_GENERAL".GENERAL_MACHINE.FROM_CELL_TO_MACHINE_GENERAL.CELL_CALIBRATION_CYCLE_REQUIRED;
   "DB426_ALARMS_WARNINGS".ALARMS.UNIT_02.STATION_3_MEASURING."720641" := #_w1;
END_REGION

REGION Network 79: UNIT 2 STATION 3 MEASURING LAST CALIBRATION OUT OF RANGE IN FIXTURE 3 ALARM
   RUNG wire#powerrail
      { S7_Templates := "SrcType := Int" } EQ_Contact(in1 := "DB16010_MEASURE_SENSORS_CALIBRATION_STATUS".U2_STA3_MEAS.FIXTURE_3_STATUS, in2 := 2)
      wire#w1
      Contact( "DB7256_UNIT_2_STA_3_MEAS_ENABLE_DISABLE".ENABLED )
      wire#w2
      I_Contact( "DB7300_INTERLOCK_GENERAL".GENERAL_MACHINE.FROM_CELL_TO_MACHINE_GENERAL.CELL_CALIBRATION_CYCLE_REQUIRED )
      Coil( "DB16000_OPC_UA_TRIGGER_ALARM".CLIENT.U2_STA3_MEAS.ALARMS.CALIBRATION_OUT_RANGE_FIX_3_A )
   END_RUNG
   RUNG wire#powerrail
      Contact( "DB16000_OPC_UA_TRIGGER_ALARM".CLIENT.U2_STA3_MEAS.ALARMS.CALIBRATION_OUT_RANGE_FIX_3_A )
      I_Contact( "DB2120_MPP_ITC_IPC".RESET_FAULTS )
   END_RUNG wire#w1
   RUNG wire#w2
      Coil( "DB426_ALARMS_WARNINGS".ALARMS.UNIT_02.STATION_3_MEASURING."720642" )
   END_RUNG
   // the same network as SCL:
   #_w1 := (("DB16010_MEASURE_SENSORS_CALIBRATION_STATUS".U2_STA3_MEAS.FIXTURE_3_STATUS = 2) OR ("DB16000_OPC_UA_TRIGGER_ALARM".CLIENT.U2_STA3_MEAS.ALARMS.CALIBRATION_OUT_RANGE_FIX_3_A AND NOT "DB2120_MPP_ITC_IPC".RESET_FAULTS)) AND "DB7256_UNIT_2_STA_3_MEAS_ENABLE_DISABLE".ENABLED;
   "DB16000_OPC_UA_TRIGGER_ALARM".CLIENT.U2_STA3_MEAS.ALARMS.CALIBRATION_OUT_RANGE_FIX_3_A := #_w1 AND NOT "DB7300_INTERLOCK_GENERAL".GENERAL_MACHINE.FROM_CELL_TO_MACHINE_GENERAL.CELL_CALIBRATION_CYCLE_REQUIRED;
   "DB426_ALARMS_WARNINGS".ALARMS.UNIT_02.STATION_3_MEASURING."720642" := #_w1;
END_REGION

REGION Network 80: UNIT 2 STATION 3 MEASURING LAST CALIBRATION OUT OF RANGE IN FIXTURE 4 ALARM
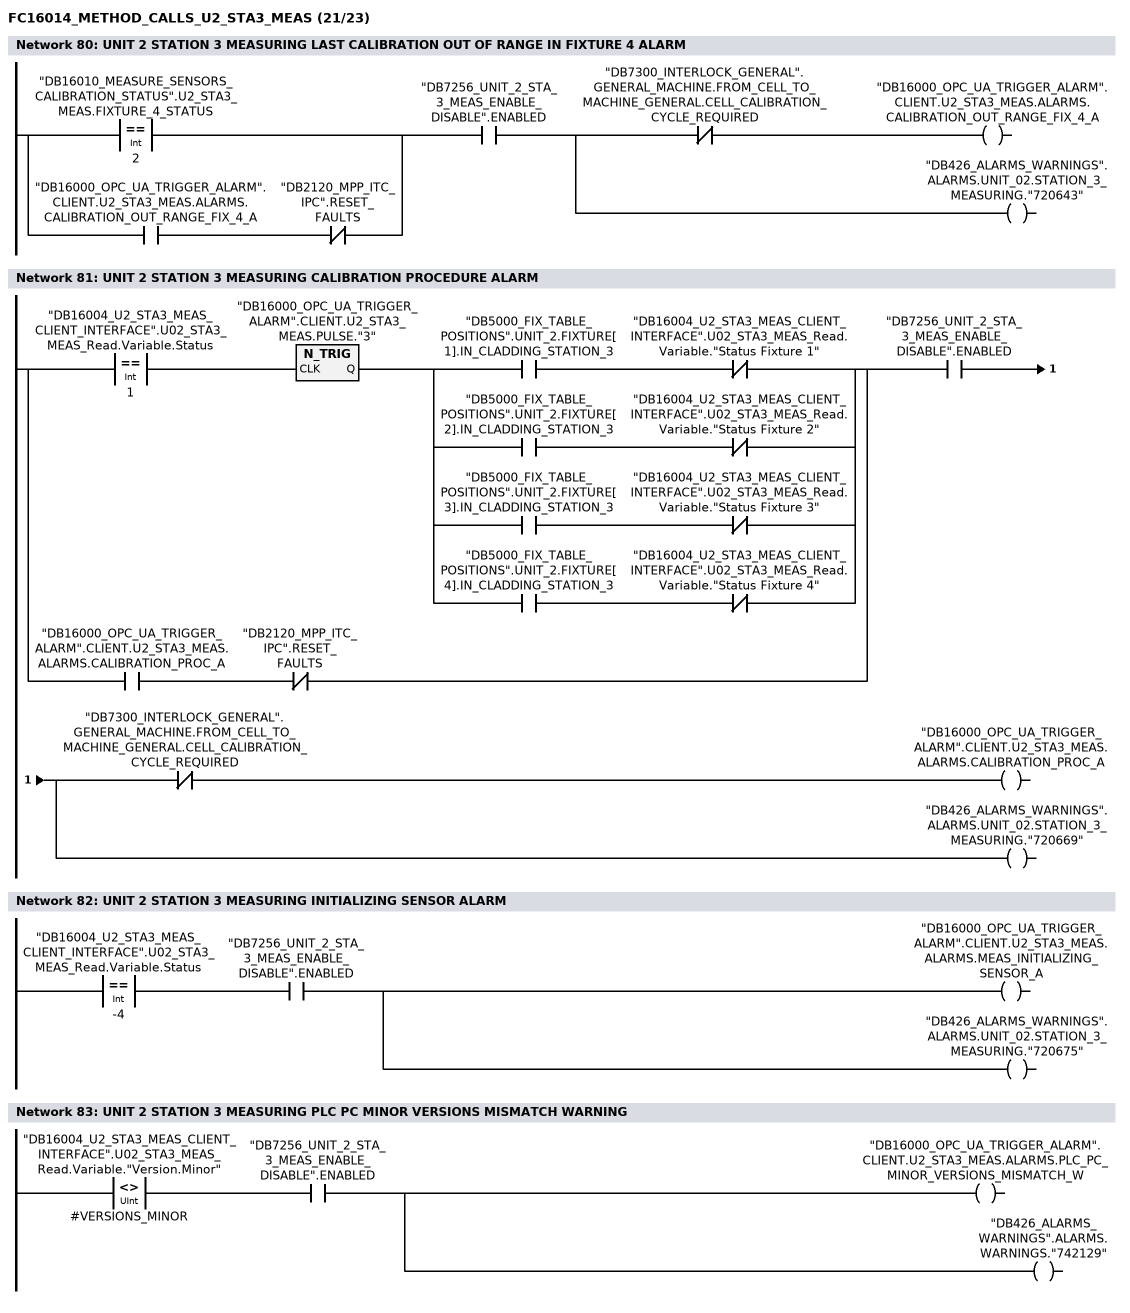
   RUNG wire#powerrail
      { S7_Templates := "SrcType := Int" } EQ_Contact(in1 := "DB16010_MEASURE_SENSORS_CALIBRATION_STATUS".U2_STA3_MEAS.FIXTURE_4_STATUS, in2 := 2)
      wire#w1
      Contact( "DB7256_UNIT_2_STA_3_MEAS_ENABLE_DISABLE".ENABLED )
      wire#w2
      I_Contact( "DB7300_INTERLOCK_GENERAL".GENERAL_MACHINE.FROM_CELL_TO_MACHINE_GENERAL.CELL_CALIBRATION_CYCLE_REQUIRED )
      Coil( "DB16000_OPC_UA_TRIGGER_ALARM".CLIENT.U2_STA3_MEAS.ALARMS.CALIBRATION_OUT_RANGE_FIX_4_A )
   END_RUNG
   RUNG wire#powerrail
      Contact( "DB16000_OPC_UA_TRIGGER_ALARM".CLIENT.U2_STA3_MEAS.ALARMS.CALIBRATION_OUT_RANGE_FIX_4_A )
      I_Contact( "DB2120_MPP_ITC_IPC".RESET_FAULTS )
   END_RUNG wire#w1
   RUNG wire#w2
      Coil( "DB426_ALARMS_WARNINGS".ALARMS.UNIT_02.STATION_3_MEASURING."720643" )
   END_RUNG
   // the same network as SCL:
   #_w1 := (("DB16010_MEASURE_SENSORS_CALIBRATION_STATUS".U2_STA3_MEAS.FIXTURE_4_STATUS = 2) OR ("DB16000_OPC_UA_TRIGGER_ALARM".CLIENT.U2_STA3_MEAS.ALARMS.CALIBRATION_OUT_RANGE_FIX_4_A AND NOT "DB2120_MPP_ITC_IPC".RESET_FAULTS)) AND "DB7256_UNIT_2_STA_3_MEAS_ENABLE_DISABLE".ENABLED;
   "DB16000_OPC_UA_TRIGGER_ALARM".CLIENT.U2_STA3_MEAS.ALARMS.CALIBRATION_OUT_RANGE_FIX_4_A := #_w1 AND NOT "DB7300_INTERLOCK_GENERAL".GENERAL_MACHINE.FROM_CELL_TO_MACHINE_GENERAL.CELL_CALIBRATION_CYCLE_REQUIRED;
   "DB426_ALARMS_WARNINGS".ALARMS.UNIT_02.STATION_3_MEASURING."720643" := #_w1;
END_REGION

REGION Network 81: UNIT 2 STATION 3 MEASURING CALIBRATION PROCEDURE ALARM
   RUNG wire#powerrail
      { S7_Templates := "SrcType := Int" } EQ_Contact(in1 := "DB16004_U2_STA3_MEAS_CLIENT_INTERFACE".U02_STA3_MEAS_Read.Variable.Status, in2 := 1)
      N_Trig( "DB16000_OPC_UA_TRIGGER_ALARM".CLIENT.U2_STA3_MEAS.PULSE."3" )
      wire#w1
      Contact( "DB5000_FIX_TABLE_POSITIONS".UNIT_2.FIXTURE[1].IN_CLADDING_STATION_3 )
      I_Contact( "DB16004_U2_STA3_MEAS_CLIENT_INTERFACE".U02_STA3_MEAS_Read.Variable."Status Fixture 1" )
      wire#w2
      Contact( "DB7256_UNIT_2_STA_3_MEAS_ENABLE_DISABLE".ENABLED )
      wire#w3
      I_Contact( "DB7300_INTERLOCK_GENERAL".GENERAL_MACHINE.FROM_CELL_TO_MACHINE_GENERAL.CELL_CALIBRATION_CYCLE_REQUIRED )
      Coil( "DB16000_OPC_UA_TRIGGER_ALARM".CLIENT.U2_STA3_MEAS.ALARMS.CALIBRATION_PROC_A )
   END_RUNG
   RUNG wire#w1
      Contact( "DB5000_FIX_TABLE_POSITIONS".UNIT_2.FIXTURE[2].IN_CLADDING_STATION_3 )
      I_Contact( "DB16004_U2_STA3_MEAS_CLIENT_INTERFACE".U02_STA3_MEAS_Read.Variable."Status Fixture 2" )
   END_RUNG wire#w2
   RUNG wire#w1
      Contact( "DB5000_FIX_TABLE_POSITIONS".UNIT_2.FIXTURE[3].IN_CLADDING_STATION_3 )
      I_Contact( "DB16004_U2_STA3_MEAS_CLIENT_INTERFACE".U02_STA3_MEAS_Read.Variable."Status Fixture 3" )
   END_RUNG wire#w2
   RUNG wire#w1
      Contact( "DB5000_FIX_TABLE_POSITIONS".UNIT_2.FIXTURE[4].IN_CLADDING_STATION_3 )
      I_Contact( "DB16004_U2_STA3_MEAS_CLIENT_INTERFACE".U02_STA3_MEAS_Read.Variable."Status Fixture 4" )
   END_RUNG wire#w2
   RUNG wire#powerrail
      Contact( "DB16000_OPC_UA_TRIGGER_ALARM".CLIENT.U2_STA3_MEAS.ALARMS.CALIBRATION_PROC_A )
      I_Contact( "DB2120_MPP_ITC_IPC".RESET_FAULTS )
   END_RUNG wire#w2
   RUNG wire#w3
      Coil( "DB426_ALARMS_WARNINGS".ALARMS.UNIT_02.STATION_3_MEASURING."720669" )
   END_RUNG
   // the same network as SCL:
   #_w1 := "DB16004_U2_STA3_MEAS_CLIENT_INTERFACE".U02_STA3_MEAS_Read.Variable.Status = 1;
   #_w2 := NOT #_w1 AND "DB16000_OPC_UA_TRIGGER_ALARM".CLIENT.U2_STA3_MEAS.PULSE."3";   // falling edge
   "DB16000_OPC_UA_TRIGGER_ALARM".CLIENT.U2_STA3_MEAS.PULSE."3" := #_w1;
   #_w3 := ((#_w2 AND (("DB5000_FIX_TABLE_POSITIONS".UNIT_2.FIXTURE[1].IN_CLADDING_STATION_3 AND NOT "DB16004_U2_STA3_MEAS_CLIENT_INTERFACE".U02_STA3_MEAS_Read.Variable."Status Fixture 1") OR ("DB5000_FIX_TABLE_POSITIONS".UNIT_2.FIXTURE[2].IN_CLADDING_STATION_3 AND NOT "DB16004_U2_STA3_MEAS_CLIENT_INTERFACE".U02_STA3_MEAS_Read.Variable."Status Fixture 2") OR ("DB5000_FIX_TABLE_POSITIONS".UNIT_2.FIXTURE[3].IN_CLADDING_STATION_3 AND NOT "DB16004_U2_STA3_MEAS_CLIENT_INTERFACE".U02_STA3_MEAS_Read.Variable."Status Fixture 3") OR ("DB5000_FIX_TABLE_POSITIONS".UNIT_2.FIXTURE[4].IN_CLADDING_STATION_3 AND NOT "DB16004_U2_STA3_MEAS_CLIENT_INTERFACE".U02_STA3_MEAS_Read.Variable."Status Fixture 4"))) OR ("DB16000_OPC_UA_TRIGGER_ALARM".CLIENT.U2_STA3_MEAS.ALARMS.CALIBRATION_PROC_A AND NOT "DB2120_MPP_ITC_IPC".RESET_FAULTS)) AND "DB7256_UNIT_2_STA_3_MEAS_ENABLE_DISABLE".ENABLED;
   "DB16000_OPC_UA_TRIGGER_ALARM".CLIENT.U2_STA3_MEAS.ALARMS.CALIBRATION_PROC_A := #_w3 AND NOT "DB7300_INTERLOCK_GENERAL".GENERAL_MACHINE.FROM_CELL_TO_MACHINE_GENERAL.CELL_CALIBRATION_CYCLE_REQUIRED;
   "DB426_ALARMS_WARNINGS".ALARMS.UNIT_02.STATION_3_MEASURING."720669" := #_w3;
END_REGION

REGION Network 82: UNIT 2 STATION 3 MEASURING INITIALIZING SENSOR ALARM
   RUNG wire#powerrail
      { S7_Templates := "SrcType := Int" } EQ_Contact(in1 := "DB16004_U2_STA3_MEAS_CLIENT_INTERFACE".U02_STA3_MEAS_Read.Variable.Status, in2 := -4)
      Contact( "DB7256_UNIT_2_STA_3_MEAS_ENABLE_DISABLE".ENABLED )
      wire#w1
      Coil( "DB16000_OPC_UA_TRIGGER_ALARM".CLIENT.U2_STA3_MEAS.ALARMS.MEAS_INITIALIZING_SENSOR_A )
   END_RUNG
   RUNG wire#w1
      Coil( "DB426_ALARMS_WARNINGS".ALARMS.UNIT_02.STATION_3_MEASURING."720675" )
   END_RUNG
   // the same network as SCL:
   "DB16000_OPC_UA_TRIGGER_ALARM".CLIENT.U2_STA3_MEAS.ALARMS.MEAS_INITIALIZING_SENSOR_A := ("DB16004_U2_STA3_MEAS_CLIENT_INTERFACE".U02_STA3_MEAS_Read.Variable.Status = (-4)) AND "DB7256_UNIT_2_STA_3_MEAS_ENABLE_DISABLE".ENABLED;
   "DB426_ALARMS_WARNINGS".ALARMS.UNIT_02.STATION_3_MEASURING."720675" := "DB16000_OPC_UA_TRIGGER_ALARM".CLIENT.U2_STA3_MEAS.ALARMS.MEAS_INITIALIZING_SENSOR_A;
END_REGION

REGION Network 83: UNIT 2 STATION 3 MEASURING PLC PC MINOR VERSIONS MISMATCH WARNING
   RUNG wire#powerrail
      { S7_Templates := "SrcType := UInt" } NE_Contact(in1 := "DB16004_U2_STA3_MEAS_CLIENT_INTERFACE".U02_STA3_MEAS_Read.Variable."Version.Minor", in2 := #VERSIONS_MINOR)
      Contact( "DB7256_UNIT_2_STA_3_MEAS_ENABLE_DISABLE".ENABLED )
      wire#w1
      Coil( "DB16000_OPC_UA_TRIGGER_ALARM".CLIENT.U2_STA3_MEAS.ALARMS.PLC_PC_MINOR_VERSIONS_MISMATCH_W )
   END_RUNG
   RUNG wire#w1
      Coil( "DB426_ALARMS_WARNINGS".ALARMS.WARNINGS."742129" )
   END_RUNG
   // the same network as SCL:
   "DB16000_OPC_UA_TRIGGER_ALARM".CLIENT.U2_STA3_MEAS.ALARMS.PLC_PC_MINOR_VERSIONS_MISMATCH_W := ("DB16004_U2_STA3_MEAS_CLIENT_INTERFACE".U02_STA3_MEAS_Read.Variable."Version.Minor" <> #VERSIONS_MINOR) AND "DB7256_UNIT_2_STA_3_MEAS_ENABLE_DISABLE".ENABLED;
   "DB426_ALARMS_WARNINGS".ALARMS.WARNINGS."742129" := "DB16000_OPC_UA_TRIGGER_ALARM".CLIENT.U2_STA3_MEAS.ALARMS.PLC_PC_MINOR_VERSIONS_MISMATCH_W;
END_REGION

REGION Network 84: UNIT 2 STATION 3 COAXIAL CAMERA PLC PC MAJOR VERSIONS MISMATCH ALARM
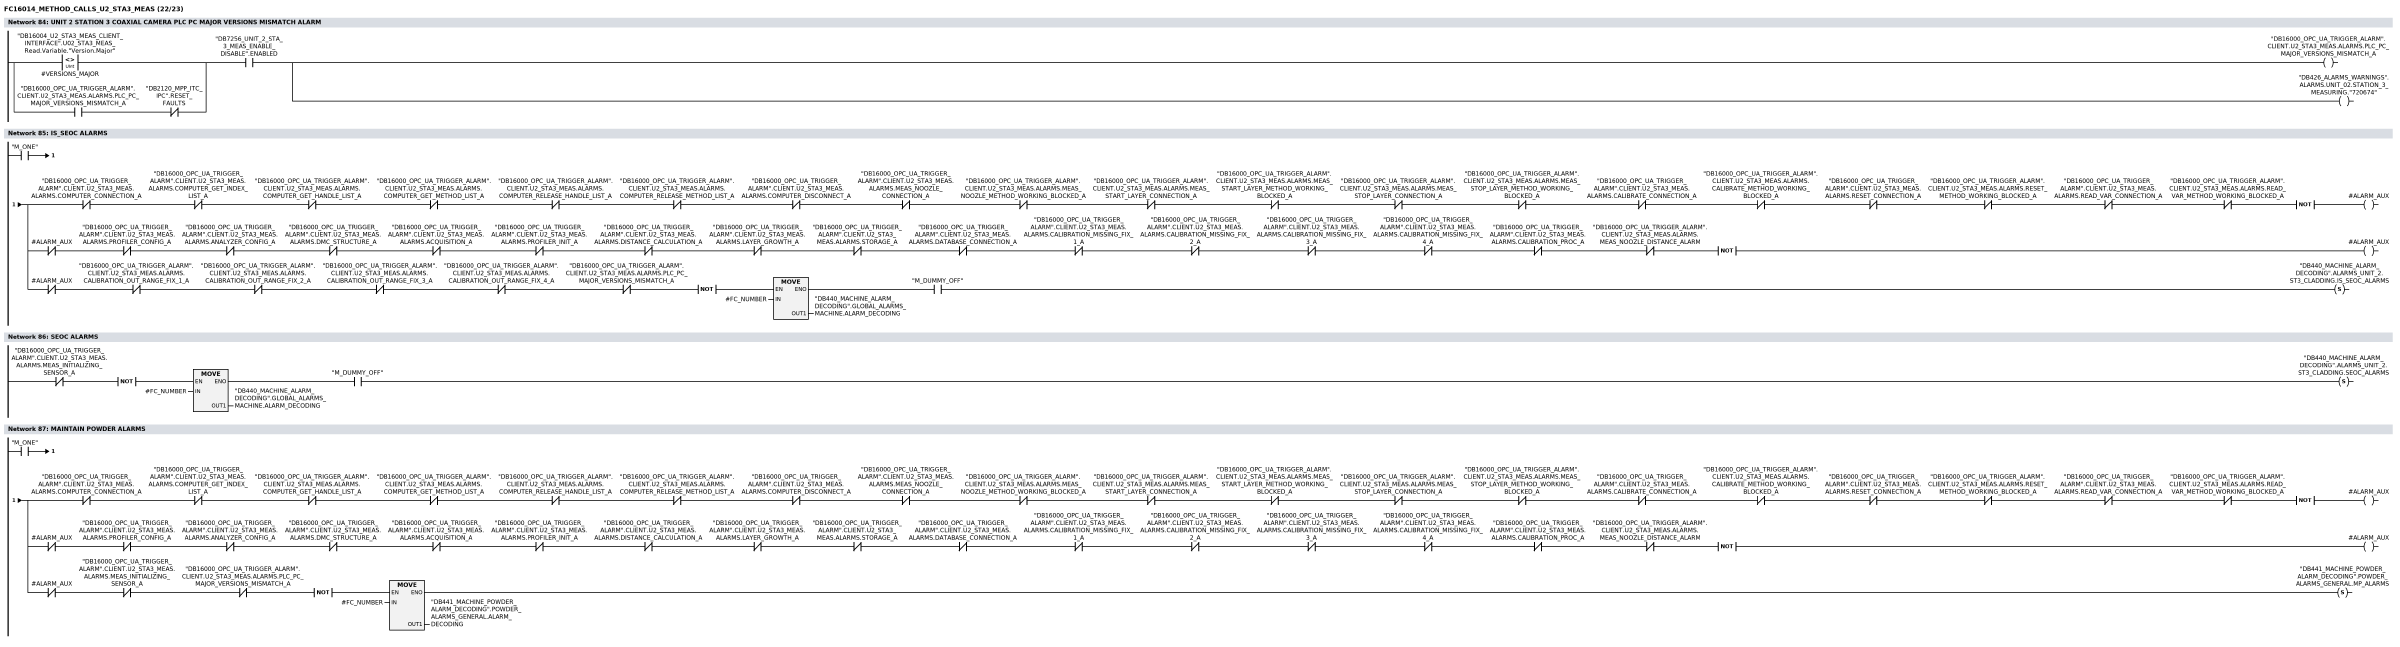
   RUNG wire#powerrail
      { S7_Templates := "SrcType := UInt" } NE_Contact(in1 := "DB16004_U2_STA3_MEAS_CLIENT_INTERFACE".U02_STA3_MEAS_Read.Variable."Version.Major", in2 := #VERSIONS_MAJOR)
      wire#w1
      Contact( "DB7256_UNIT_2_STA_3_MEAS_ENABLE_DISABLE".ENABLED )
      wire#w2
      Coil( "DB16000_OPC_UA_TRIGGER_ALARM".CLIENT.U2_STA3_MEAS.ALARMS.PLC_PC_MAJOR_VERSIONS_MISMATCH_A )
   END_RUNG
   RUNG wire#powerrail
      Contact( "DB16000_OPC_UA_TRIGGER_ALARM".CLIENT.U2_STA3_MEAS.ALARMS.PLC_PC_MAJOR_VERSIONS_MISMATCH_A )
      I_Contact( "DB2120_MPP_ITC_IPC".RESET_FAULTS )
   END_RUNG wire#w1
   RUNG wire#w2
      Coil( "DB426_ALARMS_WARNINGS".ALARMS.UNIT_02.STATION_3_MEASURING."720674" )
   END_RUNG
   // the same network as SCL:
   "DB16000_OPC_UA_TRIGGER_ALARM".CLIENT.U2_STA3_MEAS.ALARMS.PLC_PC_MAJOR_VERSIONS_MISMATCH_A := (("DB16004_U2_STA3_MEAS_CLIENT_INTERFACE".U02_STA3_MEAS_Read.Variable."Version.Major" <> #VERSIONS_MAJOR) OR ("DB16000_OPC_UA_TRIGGER_ALARM".CLIENT.U2_STA3_MEAS.ALARMS.PLC_PC_MAJOR_VERSIONS_MISMATCH_A AND NOT "DB2120_MPP_ITC_IPC".RESET_FAULTS)) AND "DB7256_UNIT_2_STA_3_MEAS_ENABLE_DISABLE".ENABLED;
   "DB426_ALARMS_WARNINGS".ALARMS.UNIT_02.STATION_3_MEASURING."720674" := "DB16000_OPC_UA_TRIGGER_ALARM".CLIENT.U2_STA3_MEAS.ALARMS.PLC_PC_MAJOR_VERSIONS_MISMATCH_A;
END_REGION

REGION Network 85: IS_SEOC ALARMS
   RUNG wire#powerrail
      Contact( "M_ONE" )
      wire#w1
      I_Contact( "DB16000_OPC_UA_TRIGGER_ALARM".CLIENT.U2_STA3_MEAS.ALARMS.COMPUTER_CONNECTION_A )
      I_Contact( "DB16000_OPC_UA_TRIGGER_ALARM".CLIENT.U2_STA3_MEAS.ALARMS.COMPUTER_GET_INDEX_LIST_A )
      I_Contact( "DB16000_OPC_UA_TRIGGER_ALARM".CLIENT.U2_STA3_MEAS.ALARMS.COMPUTER_GET_HANDLE_LIST_A )
      I_Contact( "DB16000_OPC_UA_TRIGGER_ALARM".CLIENT.U2_STA3_MEAS.ALARMS.COMPUTER_GET_METHOD_LIST_A )
      I_Contact( "DB16000_OPC_UA_TRIGGER_ALARM".CLIENT.U2_STA3_MEAS.ALARMS.COMPUTER_RELEASE_HANDLE_LIST_A )
      I_Contact( "DB16000_OPC_UA_TRIGGER_ALARM".CLIENT.U2_STA3_MEAS.ALARMS.COMPUTER_RELEASE_METHOD_LIST_A )
      I_Contact( "DB16000_OPC_UA_TRIGGER_ALARM".CLIENT.U2_STA3_MEAS.ALARMS.COMPUTER_DISCONNECT_A )
      I_Contact( "DB16000_OPC_UA_TRIGGER_ALARM".CLIENT.U2_STA3_MEAS.ALARMS.MEAS_NOOZLE_CONNECTION_A )
      I_Contact( "DB16000_OPC_UA_TRIGGER_ALARM".CLIENT.U2_STA3_MEAS.ALARMS.MEAS_NOOZLE_METHOD_WORKING_BLOCKED_A )
      I_Contact( "DB16000_OPC_UA_TRIGGER_ALARM".CLIENT.U2_STA3_MEAS.ALARMS.MEAS_START_LAYER_CONNECTION_A )
      I_Contact( "DB16000_OPC_UA_TRIGGER_ALARM".CLIENT.U2_STA3_MEAS.ALARMS.MEAS_START_LAYER_METHOD_WORKING_BLOCKED_A )
      I_Contact( "DB16000_OPC_UA_TRIGGER_ALARM".CLIENT.U2_STA3_MEAS.ALARMS.MEAS_STOP_LAYER_CONNECTION_A )
      I_Contact( "DB16000_OPC_UA_TRIGGER_ALARM".CLIENT.U2_STA3_MEAS.ALARMS.MEAS_STOP_LAYER_METHOD_WORKING_BLOCKED_A )
      I_Contact( "DB16000_OPC_UA_TRIGGER_ALARM".CLIENT.U2_STA3_MEAS.ALARMS.CALIBRATE_CONNECTION_A )
      I_Contact( "DB16000_OPC_UA_TRIGGER_ALARM".CLIENT.U2_STA3_MEAS.ALARMS.CALIBRATE_METHOD_WORKING_BLOCKED_A )
      I_Contact( "DB16000_OPC_UA_TRIGGER_ALARM".CLIENT.U2_STA3_MEAS.ALARMS.RESET_CONNECTION_A )
      I_Contact( "DB16000_OPC_UA_TRIGGER_ALARM".CLIENT.U2_STA3_MEAS.ALARMS.RESET_METHOD_WORKING_BLOCKED_A )
      I_Contact( "DB16000_OPC_UA_TRIGGER_ALARM".CLIENT.U2_STA3_MEAS.ALARMS.READ_VAR_CONNECTION_A )
      I_Contact( "DB16000_OPC_UA_TRIGGER_ALARM".CLIENT.U2_STA3_MEAS.ALARMS.READ_VAR_METHOD_WORKING_BLOCKED_A )
      Not()
      Coil( #ALARM_AUX )
   END_RUNG
   RUNG wire#w1
      I_Contact( #ALARM_AUX )
      I_Contact( "DB16000_OPC_UA_TRIGGER_ALARM".CLIENT.U2_STA3_MEAS.ALARMS.PROFILER_CONFIG_A )
      I_Contact( "DB16000_OPC_UA_TRIGGER_ALARM".CLIENT.U2_STA3_MEAS.ALARMS.ANALYZER_CONFIG_A )
      I_Contact( "DB16000_OPC_UA_TRIGGER_ALARM".CLIENT.U2_STA3_MEAS.ALARMS.DMC_STRUCTURE_A )
      I_Contact( "DB16000_OPC_UA_TRIGGER_ALARM".CLIENT.U2_STA3_MEAS.ALARMS.ACQUISITION_A )
      I_Contact( "DB16000_OPC_UA_TRIGGER_ALARM".CLIENT.U2_STA3_MEAS.ALARMS.PROFILER_INIT_A )
      I_Contact( "DB16000_OPC_UA_TRIGGER_ALARM".CLIENT.U2_STA3_MEAS.ALARMS.DISTANCE_CALCULATION_A )
      I_Contact( "DB16000_OPC_UA_TRIGGER_ALARM".CLIENT.U2_STA3_MEAS.ALARMS.LAYER_GROWTH_A )
      I_Contact( "DB16000_OPC_UA_TRIGGER_ALARM".CLIENT.U2_STA3_MEAS.ALARMS.STORAGE_A )
      I_Contact( "DB16000_OPC_UA_TRIGGER_ALARM".CLIENT.U2_STA3_MEAS.ALARMS.DATABASE_CONNECTION_A )
      I_Contact( "DB16000_OPC_UA_TRIGGER_ALARM".CLIENT.U2_STA3_MEAS.ALARMS.CALIBRATION_MISSING_FIX_1_A )
      I_Contact( "DB16000_OPC_UA_TRIGGER_ALARM".CLIENT.U2_STA3_MEAS.ALARMS.CALIBRATION_MISSING_FIX_2_A )
      I_Contact( "DB16000_OPC_UA_TRIGGER_ALARM".CLIENT.U2_STA3_MEAS.ALARMS.CALIBRATION_MISSING_FIX_3_A )
      I_Contact( "DB16000_OPC_UA_TRIGGER_ALARM".CLIENT.U2_STA3_MEAS.ALARMS.CALIBRATION_MISSING_FIX_4_A )
      I_Contact( "DB16000_OPC_UA_TRIGGER_ALARM".CLIENT.U2_STA3_MEAS.ALARMS.CALIBRATION_PROC_A )
      I_Contact( "DB16000_OPC_UA_TRIGGER_ALARM".CLIENT.U2_STA3_MEAS.ALARMS.MEAS_NOOZLE_DISTANCE_ALARM )
      Not()
      Coil( #ALARM_AUX )
   END_RUNG
   RUNG wire#w1
      I_Contact( #ALARM_AUX )
      I_Contact( "DB16000_OPC_UA_TRIGGER_ALARM".CLIENT.U2_STA3_MEAS.ALARMS.CALIBRATION_OUT_RANGE_FIX_1_A )
      I_Contact( "DB16000_OPC_UA_TRIGGER_ALARM".CLIENT.U2_STA3_MEAS.ALARMS.CALIBRATION_OUT_RANGE_FIX_2_A )
      I_Contact( "DB16000_OPC_UA_TRIGGER_ALARM".CLIENT.U2_STA3_MEAS.ALARMS.CALIBRATION_OUT_RANGE_FIX_3_A )
      I_Contact( "DB16000_OPC_UA_TRIGGER_ALARM".CLIENT.U2_STA3_MEAS.ALARMS.CALIBRATION_OUT_RANGE_FIX_4_A )
      I_Contact( "DB16000_OPC_UA_TRIGGER_ALARM".CLIENT.U2_STA3_MEAS.ALARMS.PLC_PC_MAJOR_VERSIONS_MISMATCH_A )
      Not()
      Move(in := #FC_NUMBER, out1 => "DB440_MACHINE_ALARM_DECODING".GLOBAL_ALARMS_MACHINE.ALARM_DECODING)
      Contact( "M_DUMMY_OFF" )
      S_Coil( "DB440_MACHINE_ALARM_DECODING".ALARMS_UNIT_2.ST3_CLADDING.IS_SEOC_ALARMS )
   END_RUNG
   // the same network as SCL:
   #ALARM_AUX := NOT ("M_ONE" AND NOT "DB16000_OPC_UA_TRIGGER_ALARM".CLIENT.U2_STA3_MEAS.ALARMS.COMPUTER_CONNECTION_A AND NOT "DB16000_OPC_UA_TRIGGER_ALARM".CLIENT.U2_STA3_MEAS.ALARMS.COMPUTER_GET_INDEX_LIST_A AND NOT "DB16000_OPC_UA_TRIGGER_ALARM".CLIENT.U2_STA3_MEAS.ALARMS.COMPUTER_GET_HANDLE_LIST_A AND NOT "DB16000_OPC_UA_TRIGGER_ALARM".CLIENT.U2_STA3_MEAS.ALARMS.COMPUTER_GET_METHOD_LIST_A AND NOT "DB16000_OPC_UA_TRIGGER_ALARM".CLIENT.U2_STA3_MEAS.ALARMS.COMPUTER_RELEASE_HANDLE_LIST_A AND NOT "DB16000_OPC_UA_TRIGGER_ALARM".CLIENT.U2_STA3_MEAS.ALARMS.COMPUTER_RELEASE_METHOD_LIST_A AND NOT "DB16000_OPC_UA_TRIGGER_ALARM".CLIENT.U2_STA3_MEAS.ALARMS.COMPUTER_DISCONNECT_A AND NOT "DB16000_OPC_UA_TRIGGER_ALARM".CLIENT.U2_STA3_MEAS.ALARMS.MEAS_NOOZLE_CONNECTION_A AND NOT "DB16000_OPC_UA_TRIGGER_ALARM".CLIENT.U2_STA3_MEAS.ALARMS.MEAS_NOOZLE_METHOD_WORKING_BLOCKED_A AND NOT "DB16000_OPC_UA_TRIGGER_ALARM".CLIENT.U2_STA3_MEAS.ALARMS.MEAS_START_LAYER_CONNECTION_A AND NOT "DB16000_OPC_UA_TRIGGER_ALARM".CLIENT.U2_STA3_MEAS.ALARMS.MEAS_START_LAYER_METHOD_WORKING_BLOCKED_A AND NOT "DB16000_OPC_UA_TRIGGER_ALARM".CLIENT.U2_STA3_MEAS.ALARMS.MEAS_STOP_LAYER_CONNECTION_A AND NOT "DB16000_OPC_UA_TRIGGER_ALARM".CLIENT.U2_STA3_MEAS.ALARMS.MEAS_STOP_LAYER_METHOD_WORKING_BLOCKED_A AND NOT "DB16000_OPC_UA_TRIGGER_ALARM".CLIENT.U2_STA3_MEAS.ALARMS.CALIBRATE_CONNECTION_A AND NOT "DB16000_OPC_UA_TRIGGER_ALARM".CLIENT.U2_STA3_MEAS.ALARMS.CALIBRATE_METHOD_WORKING_BLOCKED_A AND NOT "DB16000_OPC_UA_TRIGGER_ALARM".CLIENT.U2_STA3_MEAS.ALARMS.RESET_CONNECTION_A AND NOT "DB16000_OPC_UA_TRIGGER_ALARM".CLIENT.U2_STA3_MEAS.ALARMS.RESET_METHOD_WORKING_BLOCKED_A AND NOT "DB16000_OPC_UA_TRIGGER_ALARM".CLIENT.U2_STA3_MEAS.ALARMS.READ_VAR_CONNECTION_A AND NOT "DB16000_OPC_UA_TRIGGER_ALARM".CLIENT.U2_STA3_MEAS.ALARMS.READ_VAR_METHOD_WORKING_BLOCKED_A);
   #ALARM_AUX := NOT ("M_ONE" AND NOT #ALARM_AUX AND NOT "DB16000_OPC_UA_TRIGGER_ALARM".CLIENT.U2_STA3_MEAS.ALARMS.PROFILER_CONFIG_A AND NOT "DB16000_OPC_UA_TRIGGER_ALARM".CLIENT.U2_STA3_MEAS.ALARMS.ANALYZER_CONFIG_A AND NOT "DB16000_OPC_UA_TRIGGER_ALARM".CLIENT.U2_STA3_MEAS.ALARMS.DMC_STRUCTURE_A AND NOT "DB16000_OPC_UA_TRIGGER_ALARM".CLIENT.U2_STA3_MEAS.ALARMS.ACQUISITION_A AND NOT "DB16000_OPC_UA_TRIGGER_ALARM".CLIENT.U2_STA3_MEAS.ALARMS.PROFILER_INIT_A AND NOT "DB16000_OPC_UA_TRIGGER_ALARM".CLIENT.U2_STA3_MEAS.ALARMS.DISTANCE_CALCULATION_A AND NOT "DB16000_OPC_UA_TRIGGER_ALARM".CLIENT.U2_STA3_MEAS.ALARMS.LAYER_GROWTH_A AND NOT "DB16000_OPC_UA_TRIGGER_ALARM".CLIENT.U2_STA3_MEAS.ALARMS.STORAGE_A AND NOT "DB16000_OPC_UA_TRIGGER_ALARM".CLIENT.U2_STA3_MEAS.ALARMS.DATABASE_CONNECTION_A AND NOT "DB16000_OPC_UA_TRIGGER_ALARM".CLIENT.U2_STA3_MEAS.ALARMS.CALIBRATION_MISSING_FIX_1_A AND NOT "DB16000_OPC_UA_TRIGGER_ALARM".CLIENT.U2_STA3_MEAS.ALARMS.CALIBRATION_MISSING_FIX_2_A AND NOT "DB16000_OPC_UA_TRIGGER_ALARM".CLIENT.U2_STA3_MEAS.ALARMS.CALIBRATION_MISSING_FIX_3_A AND NOT "DB16000_OPC_UA_TRIGGER_ALARM".CLIENT.U2_STA3_MEAS.ALARMS.CALIBRATION_MISSING_FIX_4_A AND NOT "DB16000_OPC_UA_TRIGGER_ALARM".CLIENT.U2_STA3_MEAS.ALARMS.CALIBRATION_PROC_A AND NOT "DB16000_OPC_UA_TRIGGER_ALARM".CLIENT.U2_STA3_MEAS.ALARMS.MEAS_NOOZLE_DISTANCE_ALARM);
   #_w1 := NOT ("M_ONE" AND NOT #ALARM_AUX AND NOT "DB16000_OPC_UA_TRIGGER_ALARM".CLIENT.U2_STA3_MEAS.ALARMS.CALIBRATION_OUT_RANGE_FIX_1_A AND NOT "DB16000_OPC_UA_TRIGGER_ALARM".CLIENT.U2_STA3_MEAS.ALARMS.CALIBRATION_OUT_RANGE_FIX_2_A AND NOT "DB16000_OPC_UA_TRIGGER_ALARM".CLIENT.U2_STA3_MEAS.ALARMS.CALIBRATION_OUT_RANGE_FIX_3_A AND NOT "DB16000_OPC_UA_TRIGGER_ALARM".CLIENT.U2_STA3_MEAS.ALARMS.CALIBRATION_OUT_RANGE_FIX_4_A AND NOT "DB16000_OPC_UA_TRIGGER_ALARM".CLIENT.U2_STA3_MEAS.ALARMS.PLC_PC_MAJOR_VERSIONS_MISMATCH_A);
   IF #_w1 THEN "DB440_MACHINE_ALARM_DECODING".GLOBAL_ALARMS_MACHINE.ALARM_DECODING := #FC_NUMBER; END_IF;
   IF #_w1 AND "M_DUMMY_OFF" THEN
       "DB440_MACHINE_ALARM_DECODING".ALARMS_UNIT_2.ST3_CLADDING.IS_SEOC_ALARMS := TRUE;
   END_IF;
END_REGION

REGION Network 86: SEOC ALARMS
   RUNG wire#powerrail
      I_Contact( "DB16000_OPC_UA_TRIGGER_ALARM".CLIENT.U2_STA3_MEAS.ALARMS.MEAS_INITIALIZING_SENSOR_A )
      Not()
      Move(in := #FC_NUMBER, out1 => "DB440_MACHINE_ALARM_DECODING".GLOBAL_ALARMS_MACHINE.ALARM_DECODING)
      Contact( "M_DUMMY_OFF" )
      S_Coil( "DB440_MACHINE_ALARM_DECODING".ALARMS_UNIT_2.ST3_CLADDING.SEOC_ALARMS )
   END_RUNG
   // the same network as SCL:
   #_w1 := NOT (NOT "DB16000_OPC_UA_TRIGGER_ALARM".CLIENT.U2_STA3_MEAS.ALARMS.MEAS_INITIALIZING_SENSOR_A);
   IF #_w1 THEN "DB440_MACHINE_ALARM_DECODING".GLOBAL_ALARMS_MACHINE.ALARM_DECODING := #FC_NUMBER; END_IF;
   IF #_w1 AND "M_DUMMY_OFF" THEN
       "DB440_MACHINE_ALARM_DECODING".ALARMS_UNIT_2.ST3_CLADDING.SEOC_ALARMS := TRUE;
   END_IF;
END_REGION

REGION Network 87: MAINTAIN POWDER ALARMS
   RUNG wire#powerrail
      Contact( "M_ONE" )
      wire#w1
      I_Contact( "DB16000_OPC_UA_TRIGGER_ALARM".CLIENT.U2_STA3_MEAS.ALARMS.COMPUTER_CONNECTION_A )
      I_Contact( "DB16000_OPC_UA_TRIGGER_ALARM".CLIENT.U2_STA3_MEAS.ALARMS.COMPUTER_GET_INDEX_LIST_A )
      I_Contact( "DB16000_OPC_UA_TRIGGER_ALARM".CLIENT.U2_STA3_MEAS.ALARMS.COMPUTER_GET_HANDLE_LIST_A )
      I_Contact( "DB16000_OPC_UA_TRIGGER_ALARM".CLIENT.U2_STA3_MEAS.ALARMS.COMPUTER_GET_METHOD_LIST_A )
      I_Contact( "DB16000_OPC_UA_TRIGGER_ALARM".CLIENT.U2_STA3_MEAS.ALARMS.COMPUTER_RELEASE_HANDLE_LIST_A )
      I_Contact( "DB16000_OPC_UA_TRIGGER_ALARM".CLIENT.U2_STA3_MEAS.ALARMS.COMPUTER_RELEASE_METHOD_LIST_A )
      I_Contact( "DB16000_OPC_UA_TRIGGER_ALARM".CLIENT.U2_STA3_MEAS.ALARMS.COMPUTER_DISCONNECT_A )
      I_Contact( "DB16000_OPC_UA_TRIGGER_ALARM".CLIENT.U2_STA3_MEAS.ALARMS.MEAS_NOOZLE_CONNECTION_A )
      I_Contact( "DB16000_OPC_UA_TRIGGER_ALARM".CLIENT.U2_STA3_MEAS.ALARMS.MEAS_NOOZLE_METHOD_WORKING_BLOCKED_A )
      I_Contact( "DB16000_OPC_UA_TRIGGER_ALARM".CLIENT.U2_STA3_MEAS.ALARMS.MEAS_START_LAYER_CONNECTION_A )
      I_Contact( "DB16000_OPC_UA_TRIGGER_ALARM".CLIENT.U2_STA3_MEAS.ALARMS.MEAS_START_LAYER_METHOD_WORKING_BLOCKED_A )
      I_Contact( "DB16000_OPC_UA_TRIGGER_ALARM".CLIENT.U2_STA3_MEAS.ALARMS.MEAS_STOP_LAYER_CONNECTION_A )
      I_Contact( "DB16000_OPC_UA_TRIGGER_ALARM".CLIENT.U2_STA3_MEAS.ALARMS.MEAS_STOP_LAYER_METHOD_WORKING_BLOCKED_A )
      I_Contact( "DB16000_OPC_UA_TRIGGER_ALARM".CLIENT.U2_STA3_MEAS.ALARMS.CALIBRATE_CONNECTION_A )
      I_Contact( "DB16000_OPC_UA_TRIGGER_ALARM".CLIENT.U2_STA3_MEAS.ALARMS.CALIBRATE_METHOD_WORKING_BLOCKED_A )
      I_Contact( "DB16000_OPC_UA_TRIGGER_ALARM".CLIENT.U2_STA3_MEAS.ALARMS.RESET_CONNECTION_A )
      I_Contact( "DB16000_OPC_UA_TRIGGER_ALARM".CLIENT.U2_STA3_MEAS.ALARMS.RESET_METHOD_WORKING_BLOCKED_A )
      I_Contact( "DB16000_OPC_UA_TRIGGER_ALARM".CLIENT.U2_STA3_MEAS.ALARMS.READ_VAR_CONNECTION_A )
      I_Contact( "DB16000_OPC_UA_TRIGGER_ALARM".CLIENT.U2_STA3_MEAS.ALARMS.READ_VAR_METHOD_WORKING_BLOCKED_A )
      Not()
      Coil( #ALARM_AUX )
   END_RUNG
   RUNG wire#w1
      I_Contact( #ALARM_AUX )
      I_Contact( "DB16000_OPC_UA_TRIGGER_ALARM".CLIENT.U2_STA3_MEAS.ALARMS.PROFILER_CONFIG_A )
      I_Contact( "DB16000_OPC_UA_TRIGGER_ALARM".CLIENT.U2_STA3_MEAS.ALARMS.ANALYZER_CONFIG_A )
      I_Contact( "DB16000_OPC_UA_TRIGGER_ALARM".CLIENT.U2_STA3_MEAS.ALARMS.DMC_STRUCTURE_A )
      I_Contact( "DB16000_OPC_UA_TRIGGER_ALARM".CLIENT.U2_STA3_MEAS.ALARMS.ACQUISITION_A )
      I_Contact( "DB16000_OPC_UA_TRIGGER_ALARM".CLIENT.U2_STA3_MEAS.ALARMS.PROFILER_INIT_A )
      I_Contact( "DB16000_OPC_UA_TRIGGER_ALARM".CLIENT.U2_STA3_MEAS.ALARMS.DISTANCE_CALCULATION_A )
      I_Contact( "DB16000_OPC_UA_TRIGGER_ALARM".CLIENT.U2_STA3_MEAS.ALARMS.LAYER_GROWTH_A )
      I_Contact( "DB16000_OPC_UA_TRIGGER_ALARM".CLIENT.U2_STA3_MEAS.ALARMS.STORAGE_A )
      I_Contact( "DB16000_OPC_UA_TRIGGER_ALARM".CLIENT.U2_STA3_MEAS.ALARMS.DATABASE_CONNECTION_A )
      I_Contact( "DB16000_OPC_UA_TRIGGER_ALARM".CLIENT.U2_STA3_MEAS.ALARMS.CALIBRATION_MISSING_FIX_1_A )
      I_Contact( "DB16000_OPC_UA_TRIGGER_ALARM".CLIENT.U2_STA3_MEAS.ALARMS.CALIBRATION_MISSING_FIX_2_A )
      I_Contact( "DB16000_OPC_UA_TRIGGER_ALARM".CLIENT.U2_STA3_MEAS.ALARMS.CALIBRATION_MISSING_FIX_3_A )
      I_Contact( "DB16000_OPC_UA_TRIGGER_ALARM".CLIENT.U2_STA3_MEAS.ALARMS.CALIBRATION_MISSING_FIX_4_A )
      I_Contact( "DB16000_OPC_UA_TRIGGER_ALARM".CLIENT.U2_STA3_MEAS.ALARMS.CALIBRATION_PROC_A )
      I_Contact( "DB16000_OPC_UA_TRIGGER_ALARM".CLIENT.U2_STA3_MEAS.ALARMS.MEAS_NOOZLE_DISTANCE_ALARM )
      Not()
      Coil( #ALARM_AUX )
   END_RUNG
   RUNG wire#w1
      I_Contact( #ALARM_AUX )
      I_Contact( "DB16000_OPC_UA_TRIGGER_ALARM".CLIENT.U2_STA3_MEAS.ALARMS.MEAS_INITIALIZING_SENSOR_A )
      I_Contact( "DB16000_OPC_UA_TRIGGER_ALARM".CLIENT.U2_STA3_MEAS.ALARMS.PLC_PC_MAJOR_VERSIONS_MISMATCH_A )
      Not()
      Move(in := #FC_NUMBER, out1 => "DB441_MACHINE_POWDER_ALARM_DECODING".POWDER_ALARMS_GENERAL.ALARM_DECODING)
      S_Coil( "DB441_MACHINE_POWDER_ALARM_DECODING".POWDER_ALARMS_GENERAL.MP_ALARMS )
   END_RUNG
   // the same network as SCL:
   #ALARM_AUX := NOT ("M_ONE" AND NOT "DB16000_OPC_UA_TRIGGER_ALARM".CLIENT.U2_STA3_MEAS.ALARMS.COMPUTER_CONNECTION_A AND NOT "DB16000_OPC_UA_TRIGGER_ALARM".CLIENT.U2_STA3_MEAS.ALARMS.COMPUTER_GET_INDEX_LIST_A AND NOT "DB16000_OPC_UA_TRIGGER_ALARM".CLIENT.U2_STA3_MEAS.ALARMS.COMPUTER_GET_HANDLE_LIST_A AND NOT "DB16000_OPC_UA_TRIGGER_ALARM".CLIENT.U2_STA3_MEAS.ALARMS.COMPUTER_GET_METHOD_LIST_A AND NOT "DB16000_OPC_UA_TRIGGER_ALARM".CLIENT.U2_STA3_MEAS.ALARMS.COMPUTER_RELEASE_HANDLE_LIST_A AND NOT "DB16000_OPC_UA_TRIGGER_ALARM".CLIENT.U2_STA3_MEAS.ALARMS.COMPUTER_RELEASE_METHOD_LIST_A AND NOT "DB16000_OPC_UA_TRIGGER_ALARM".CLIENT.U2_STA3_MEAS.ALARMS.COMPUTER_DISCONNECT_A AND NOT "DB16000_OPC_UA_TRIGGER_ALARM".CLIENT.U2_STA3_MEAS.ALARMS.MEAS_NOOZLE_CONNECTION_A AND NOT "DB16000_OPC_UA_TRIGGER_ALARM".CLIENT.U2_STA3_MEAS.ALARMS.MEAS_NOOZLE_METHOD_WORKING_BLOCKED_A AND NOT "DB16000_OPC_UA_TRIGGER_ALARM".CLIENT.U2_STA3_MEAS.ALARMS.MEAS_START_LAYER_CONNECTION_A AND NOT "DB16000_OPC_UA_TRIGGER_ALARM".CLIENT.U2_STA3_MEAS.ALARMS.MEAS_START_LAYER_METHOD_WORKING_BLOCKED_A AND NOT "DB16000_OPC_UA_TRIGGER_ALARM".CLIENT.U2_STA3_MEAS.ALARMS.MEAS_STOP_LAYER_CONNECTION_A AND NOT "DB16000_OPC_UA_TRIGGER_ALARM".CLIENT.U2_STA3_MEAS.ALARMS.MEAS_STOP_LAYER_METHOD_WORKING_BLOCKED_A AND NOT "DB16000_OPC_UA_TRIGGER_ALARM".CLIENT.U2_STA3_MEAS.ALARMS.CALIBRATE_CONNECTION_A AND NOT "DB16000_OPC_UA_TRIGGER_ALARM".CLIENT.U2_STA3_MEAS.ALARMS.CALIBRATE_METHOD_WORKING_BLOCKED_A AND NOT "DB16000_OPC_UA_TRIGGER_ALARM".CLIENT.U2_STA3_MEAS.ALARMS.RESET_CONNECTION_A AND NOT "DB16000_OPC_UA_TRIGGER_ALARM".CLIENT.U2_STA3_MEAS.ALARMS.RESET_METHOD_WORKING_BLOCKED_A AND NOT "DB16000_OPC_UA_TRIGGER_ALARM".CLIENT.U2_STA3_MEAS.ALARMS.READ_VAR_CONNECTION_A AND NOT "DB16000_OPC_UA_TRIGGER_ALARM".CLIENT.U2_STA3_MEAS.ALARMS.READ_VAR_METHOD_WORKING_BLOCKED_A);
   #ALARM_AUX := NOT ("M_ONE" AND NOT #ALARM_AUX AND NOT "DB16000_OPC_UA_TRIGGER_ALARM".CLIENT.U2_STA3_MEAS.ALARMS.PROFILER_CONFIG_A AND NOT "DB16000_OPC_UA_TRIGGER_ALARM".CLIENT.U2_STA3_MEAS.ALARMS.ANALYZER_CONFIG_A AND NOT "DB16000_OPC_UA_TRIGGER_ALARM".CLIENT.U2_STA3_MEAS.ALARMS.DMC_STRUCTURE_A AND NOT "DB16000_OPC_UA_TRIGGER_ALARM".CLIENT.U2_STA3_MEAS.ALARMS.ACQUISITION_A AND NOT "DB16000_OPC_UA_TRIGGER_ALARM".CLIENT.U2_STA3_MEAS.ALARMS.PROFILER_INIT_A AND NOT "DB16000_OPC_UA_TRIGGER_ALARM".CLIENT.U2_STA3_MEAS.ALARMS.DISTANCE_CALCULATION_A AND NOT "DB16000_OPC_UA_TRIGGER_ALARM".CLIENT.U2_STA3_MEAS.ALARMS.LAYER_GROWTH_A AND NOT "DB16000_OPC_UA_TRIGGER_ALARM".CLIENT.U2_STA3_MEAS.ALARMS.STORAGE_A AND NOT "DB16000_OPC_UA_TRIGGER_ALARM".CLIENT.U2_STA3_MEAS.ALARMS.DATABASE_CONNECTION_A AND NOT "DB16000_OPC_UA_TRIGGER_ALARM".CLIENT.U2_STA3_MEAS.ALARMS.CALIBRATION_MISSING_FIX_1_A AND NOT "DB16000_OPC_UA_TRIGGER_ALARM".CLIENT.U2_STA3_MEAS.ALARMS.CALIBRATION_MISSING_FIX_2_A AND NOT "DB16000_OPC_UA_TRIGGER_ALARM".CLIENT.U2_STA3_MEAS.ALARMS.CALIBRATION_MISSING_FIX_3_A AND NOT "DB16000_OPC_UA_TRIGGER_ALARM".CLIENT.U2_STA3_MEAS.ALARMS.CALIBRATION_MISSING_FIX_4_A AND NOT "DB16000_OPC_UA_TRIGGER_ALARM".CLIENT.U2_STA3_MEAS.ALARMS.CALIBRATION_PROC_A AND NOT "DB16000_OPC_UA_TRIGGER_ALARM".CLIENT.U2_STA3_MEAS.ALARMS.MEAS_NOOZLE_DISTANCE_ALARM);
   IF NOT ("M_ONE" AND NOT #ALARM_AUX AND NOT "DB16000_OPC_UA_TRIGGER_ALARM".CLIENT.U2_STA3_MEAS.ALARMS.MEAS_INITIALIZING_SENSOR_A AND NOT "DB16000_OPC_UA_TRIGGER_ALARM".CLIENT.U2_STA3_MEAS.ALARMS.PLC_PC_MAJOR_VERSIONS_MISMATCH_A) THEN
       "DB441_MACHINE_POWDER_ALARM_DECODING".POWDER_ALARMS_GENERAL.ALARM_DECODING := #FC_NUMBER;
       "DB441_MACHINE_POWDER_ALARM_DECODING".POWDER_ALARMS_GENERAL.MP_ALARMS := TRUE;
   END_IF;
END_REGION

REGION Network 88: PROGRESSIVE STOP POWDER ALARMS
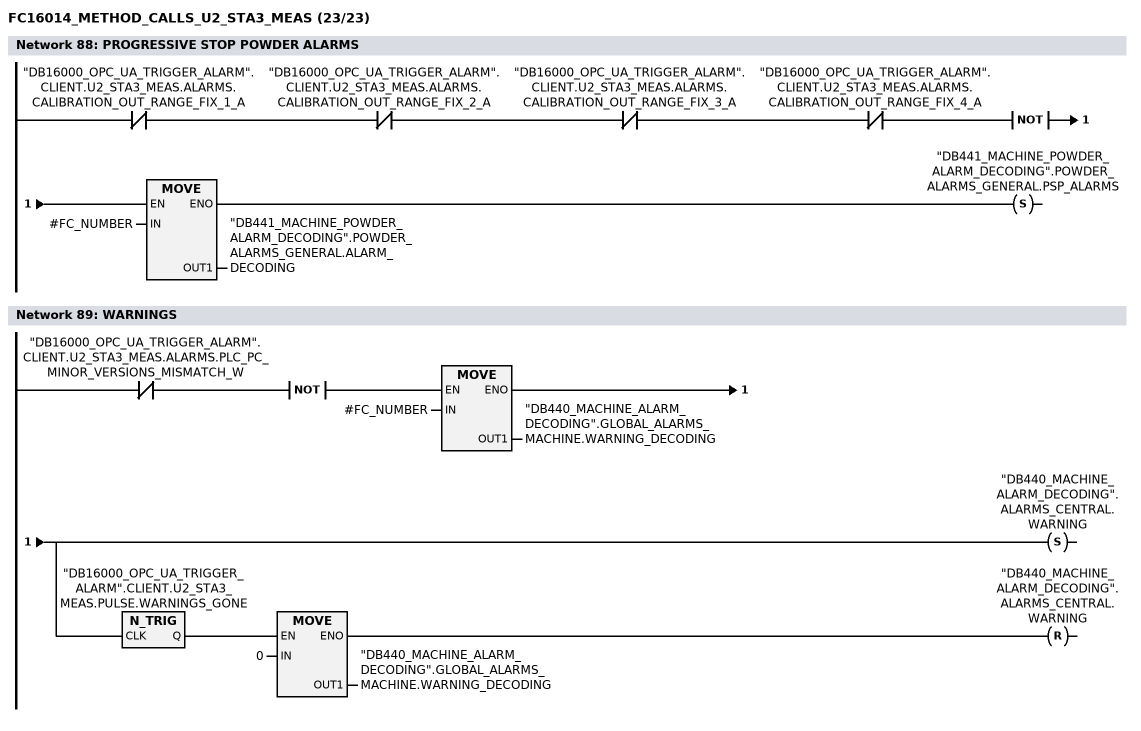
   RUNG wire#powerrail
      I_Contact( "DB16000_OPC_UA_TRIGGER_ALARM".CLIENT.U2_STA3_MEAS.ALARMS.CALIBRATION_OUT_RANGE_FIX_1_A )
      I_Contact( "DB16000_OPC_UA_TRIGGER_ALARM".CLIENT.U2_STA3_MEAS.ALARMS.CALIBRATION_OUT_RANGE_FIX_2_A )
      I_Contact( "DB16000_OPC_UA_TRIGGER_ALARM".CLIENT.U2_STA3_MEAS.ALARMS.CALIBRATION_OUT_RANGE_FIX_3_A )
      I_Contact( "DB16000_OPC_UA_TRIGGER_ALARM".CLIENT.U2_STA3_MEAS.ALARMS.CALIBRATION_OUT_RANGE_FIX_4_A )
      Not()
      Move(in := #FC_NUMBER, out1 => "DB441_MACHINE_POWDER_ALARM_DECODING".POWDER_ALARMS_GENERAL.ALARM_DECODING)
      S_Coil( "DB441_MACHINE_POWDER_ALARM_DECODING".POWDER_ALARMS_GENERAL.PSP_ALARMS )
   END_RUNG
   // the same network as SCL:
   IF NOT (NOT "DB16000_OPC_UA_TRIGGER_ALARM".CLIENT.U2_STA3_MEAS.ALARMS.CALIBRATION_OUT_RANGE_FIX_1_A AND NOT "DB16000_OPC_UA_TRIGGER_ALARM".CLIENT.U2_STA3_MEAS.ALARMS.CALIBRATION_OUT_RANGE_FIX_2_A AND NOT "DB16000_OPC_UA_TRIGGER_ALARM".CLIENT.U2_STA3_MEAS.ALARMS.CALIBRATION_OUT_RANGE_FIX_3_A AND NOT "DB16000_OPC_UA_TRIGGER_ALARM".CLIENT.U2_STA3_MEAS.ALARMS.CALIBRATION_OUT_RANGE_FIX_4_A) THEN
       "DB441_MACHINE_POWDER_ALARM_DECODING".POWDER_ALARMS_GENERAL.ALARM_DECODING := #FC_NUMBER;
       "DB441_MACHINE_POWDER_ALARM_DECODING".POWDER_ALARMS_GENERAL.PSP_ALARMS := TRUE;
   END_IF;
END_REGION

REGION Network 89: WARNINGS
   RUNG wire#powerrail
      I_Contact( "DB16000_OPC_UA_TRIGGER_ALARM".CLIENT.U2_STA3_MEAS.ALARMS.PLC_PC_MINOR_VERSIONS_MISMATCH_W )
      Not()
      Move(in := #FC_NUMBER, out1 => "DB440_MACHINE_ALARM_DECODING".GLOBAL_ALARMS_MACHINE.WARNING_DECODING)
      wire#w1
      S_Coil( "DB440_MACHINE_ALARM_DECODING".ALARMS_CENTRAL.WARNING )
   END_RUNG
   RUNG wire#w1
      N_Trig( "DB16000_OPC_UA_TRIGGER_ALARM".CLIENT.U2_STA3_MEAS.PULSE.WARNINGS_GONE )
      Move(in := 0, out1 => "DB440_MACHINE_ALARM_DECODING".GLOBAL_ALARMS_MACHINE.WARNING_DECODING)
      R_Coil( "DB440_MACHINE_ALARM_DECODING".ALARMS_CENTRAL.WARNING )
   END_RUNG
   // the same network as SCL:
   #_w1 := NOT (NOT "DB16000_OPC_UA_TRIGGER_ALARM".CLIENT.U2_STA3_MEAS.ALARMS.PLC_PC_MINOR_VERSIONS_MISMATCH_W);
   IF #_w1 THEN
       "DB440_MACHINE_ALARM_DECODING".GLOBAL_ALARMS_MACHINE.WARNING_DECODING := #FC_NUMBER;
       "DB440_MACHINE_ALARM_DECODING".ALARMS_CENTRAL.WARNING := TRUE;
   END_IF;
   #_w2 := NOT #_w1 AND "DB16000_OPC_UA_TRIGGER_ALARM".CLIENT.U2_STA3_MEAS.PULSE.WARNINGS_GONE;   // falling edge
   "DB16000_OPC_UA_TRIGGER_ALARM".CLIENT.U2_STA3_MEAS.PULSE.WARNINGS_GONE := #_w1;
   IF #_w2 THEN
       "DB440_MACHINE_ALARM_DECODING".GLOBAL_ALARMS_MACHINE.WARNING_DECODING := 0;
       "DB440_MACHINE_ALARM_DECODING".ALARMS_CENTRAL.WARNING := FALSE;
   END_IF;
END_REGION
END_FUNCTION
